   LIN {X -6.651, Y 41.522, Z 66.300}
   LaserStart_Ext()
   LIN {X -0.584, Y 41.522, Z 66.300}
   LaserEnd_Ext()
   LIN {X -0.132, Y 40.522, Z 66.300}
   LaserStart_Ext()
   LIN {X -6.592, Y 40.522, Z 66.300}
   LaserEnd_Ext()
   LIN {X -6.269, Y 39.522, Z 66.300}
   LaserStart_Ext()
   LIN {X 0.315, Y 39.522, Z 66.300}
   LaserEnd_Ext()
   LIN {X 0.738, Y 38.522, Z 66.300}
   LaserStart_Ext()
   LIN {X -5.884, Y 38.522, Z 66.300}
   LaserEnd_Ext()
   LIN {X -5.510, Y 37.522, Z 66.300}
   LaserStart_Ext()
   LIN {X 1.160, Y 37.522, Z 66.300}
   LaserEnd_Ext()
   LIN {X 1.563, Y 36.522, Z 66.300}
   LaserStart_Ext()
   LIN {X -5.164, Y 36.522, Z 66.300}
   LaserEnd_Ext()
   LIN {X -4.819, Y 35.522, Z 66.300}
   LaserStart_Ext()
   LIN {X 1.943, Y 35.522, Z 66.300}
   LaserEnd_Ext()
   LIN {X 2.327, Y 34.522, Z 66.300}
   LaserStart_Ext()
   LIN {X -4.502, Y 34.522, Z 66.300}
   LaserEnd_Ext()
   LIN {X -4.196, Y 33.522, Z 66.300}
   LaserStart_Ext()
   LIN {X 2.711, Y 33.522, Z 66.300}
   LaserEnd_Ext()
   LIN {X 3.089, Y 32.522, Z 66.300}
   LaserStart_Ext()
   LIN {X -3.888, Y 32.522, Z 66.300}
   LaserEnd_Ext()
   LIN {X -3.629, Y 31.522, Z 66.300}
   LaserStart_Ext()
   LIN {X 3.434, Y 31.522, Z 66.300}
   LaserEnd_Ext()
   LIN {X 3.759, Y 30.522, Z 66.300}
   LaserStart_Ext()
   LIN {X -3.371, Y 30.522, Z 66.300}
   LaserEnd_Ext()
   LIN {X -3.113, Y 29.522, Z 66.300}
   LaserStart_Ext()
   LIN {X 4.082, Y 29.522, Z 66.300}
   LaserEnd_Ext()
   LIN {X 4.405, Y 28.522, Z 66.300}
   LaserStart_Ext()
   LIN {X -2.876, Y 28.522, Z 66.300}
   LaserEnd_Ext()
   LIN {X -2.680, Y 27.522, Z 66.300}
   LaserStart_Ext()
   LIN {X 4.728, Y 27.522, Z 66.300}
   LaserEnd_Ext()
   LIN {X 5.051, Y 26.522, Z 66.300}
   LaserStart_Ext()
   LIN {X -2.482, Y 26.522, Z 66.300}
   LaserEnd_Ext()
   LIN {X -2.285, Y 25.522, Z 66.300}
   LaserStart_Ext()
   LIN {X 5.305, Y 25.522, Z 66.300}
   LaserEnd_Ext()
   LIN {X 5.559, Y 24.522, Z 66.300}
   LaserStart_Ext()
   LIN {X -2.087, Y 24.522, Z 66.300}
   LaserEnd_Ext()
   LIN {X -1.950, Y 23.522, Z 66.300}
   LaserStart_Ext()
   LIN {X 5.812, Y 23.522, Z 66.300}
   LaserEnd_Ext()
   LIN {X 6.066, Y 22.522, Z 66.300}
   LaserStart_Ext()
   LIN {X -1.864, Y 22.522, Z 66.300}
   LaserEnd_Ext()
   LIN {X -1.779, Y 21.522, Z 66.300}
   LaserStart_Ext()
   LIN {X 6.319, Y 21.522, Z 66.300}
   LaserEnd_Ext()
   LIN {X 6.573, Y 20.522, Z 66.300}
   LaserStart_Ext()
   LIN {X -1.694, Y 20.522, Z 66.300}
   LaserEnd_Ext()
   LIN {X -1.588, Y 19.522, Z 66.300}
   LaserStart_Ext()
   LIN {X 6.833, Y 19.522, Z 66.300}
   LaserEnd_Ext()
   LIN {X 7.071, Y 18.522, Z 66.300}
   LaserStart_Ext()
   LIN {X -1.481, Y 18.522, Z 66.300}
   LaserEnd_Ext()
   LIN {X -1.375, Y 17.522, Z 66.300}
   LaserStart_Ext()
   LIN {X 7.250, Y 17.522, Z 66.300}
   LaserEnd_Ext()
   LIN {X 7.405, Y 16.522, Z 66.300}
   LaserStart_Ext()
   LIN {X -1.269, Y 16.522, Z 66.300}
   LaserEnd_Ext()
   LIN {X -1.163, Y 15.522, Z 66.300}
   LaserStart_Ext()
   LIN {X 7.561, Y 15.522, Z 66.300}
   LaserEnd_Ext()
   LIN {X 7.716, Y 14.522, Z 66.300}
   LaserStart_Ext()
   LIN {X -1.142, Y 14.522, Z 66.300}
   LaserEnd_Ext()
   LIN {X -1.150, Y 13.522, Z 66.300}
   LaserStart_Ext()
   LIN {X 7.872, Y 13.522, Z 66.300}
   LaserEnd_Ext()
   LIN {X 8.027, Y 12.522, Z 66.300}
   LaserStart_Ext()
   LIN {X -1.158, Y 12.522, Z 66.300}
   LaserEnd_Ext()
   LIN {X -1.166, Y 11.522, Z 66.300}
   LaserStart_Ext()
   LIN {X 8.183, Y 11.522, Z 66.300}
   LaserEnd_Ext()
   LIN {X 8.339, Y 10.522, Z 66.300}
   LaserStart_Ext()
   LIN {X -1.175, Y 10.522, Z 66.300}
   LaserEnd_Ext()
   LIN {X -1.191, Y 9.522, Z 66.300}
   LaserStart_Ext()
   LIN {X 8.494, Y 9.522, Z 66.300}
   LaserEnd_Ext()
   LIN {X 8.650, Y 8.522, Z 66.300}
   LaserStart_Ext()
   LIN {X -1.230, Y 8.522, Z 66.300}
   LaserEnd_Ext()
   LIN {X -1.268, Y 7.522, Z 66.300}
   LaserStart_Ext()
   LIN {X 8.806, Y 7.522, Z 66.300}
   LaserEnd_Ext()
   LIN {X 8.956, Y 6.522, Z 66.300}
   LaserStart_Ext()
   LIN {X -1.307, Y 6.522, Z 66.300}
   LaserEnd_Ext()
   LIN {X -1.345, Y 5.522, Z 66.300}
   LaserStart_Ext()
   LIN {X 9.069, Y 5.522, Z 66.300}
   LaserEnd_Ext()
   LIN {X 9.141, Y 4.522, Z 66.300}
   LaserStart_Ext()
   LIN {X -1.463, Y 4.522, Z 66.300}
   LaserEnd_Ext()
   LIN {X -1.598, Y 3.522, Z 66.300}
   LaserStart_Ext()
   LIN {X 9.202, Y 3.522, Z 66.300}
   LaserEnd_Ext()
   LIN {X 9.264, Y 2.522, Z 66.300}
   LaserStart_Ext()
   LIN {X -1.733, Y 2.522, Z 66.300}
   LaserEnd_Ext()
   LIN {X -1.868, Y 1.522, Z 66.300}
   LaserStart_Ext()
   LIN {X 9.325, Y 1.522, Z 66.300}
   LaserEnd_Ext()
   LIN {X 9.387, Y 0.522, Z 66.300}
   LaserStart_Ext()
   LIN {X -2.004, Y 0.522, Z 66.300}
   LaserEnd_Ext()
   LIN {X -2.141, Y -0.478, Z 66.300}
   LaserStart_Ext()
   LIN {X 9.437, Y -0.478, Z 66.300}
   LaserEnd_Ext()
   LIN {X 9.443, Y -1.478, Z 66.300}
   LaserStart_Ext()
   LIN {X -2.360, Y -1.478, Z 66.300}
   LaserEnd_Ext()
   LIN {X -2.584, Y -2.478, Z 66.300}
   LaserStart_Ext()
   LIN {X 9.450, Y -2.478, Z 66.300}
   LaserEnd_Ext()
   LIN {X 9.459, Y -3.478, Z 66.300}
   LaserStart_Ext()
   LIN {X -2.803, Y -3.478, Z 66.300}
   LaserEnd_Ext()
   LIN {X -3.022, Y -4.478, Z 66.300}
   LaserStart_Ext()
   LIN {X 9.468, Y -4.478, Z 66.300}
   LaserEnd_Ext()
   LIN {X 9.477, Y -5.478, Z 66.300}
   LaserStart_Ext()
   LIN {X -3.241, Y -5.478, Z 66.300}
   LaserEnd_Ext()
   LIN {X -3.460, Y -6.478, Z 66.300}
   LaserStart_Ext()
   LIN {X 9.486, Y -6.478, Z 66.300}
   LaserEnd_Ext()
   LIN {X 9.460, Y -7.478, Z 66.300}
   LaserStart_Ext()
   LIN {X -3.732, Y -7.478, Z 66.300}
   LaserEnd_Ext()
   LIN {X -4.029, Y -8.478, Z 66.300}
   LaserStart_Ext()
   LIN {X 9.419, Y -8.478, Z 66.300}
   LaserEnd_Ext()
   LIN {X 9.374, Y -9.478, Z 66.300}
   LaserStart_Ext()
   LIN {X -4.322, Y -9.478, Z 66.300}
   LaserEnd_Ext()
   LIN {X -4.616, Y -10.478, Z 66.300}
   LaserStart_Ext()
   LIN {X 9.329, Y -10.478, Z 66.300}
   LaserEnd_Ext()
   LIN {X 9.284, Y -11.478, Z 66.300}
   LaserStart_Ext()
   LIN {X -4.963, Y -11.478, Z 66.300}
   LaserEnd_Ext()
   LIN {X -5.315, Y -12.478, Z 66.300}
   LaserStart_Ext()
   LIN {X 9.205, Y -12.478, Z 66.300}
   LaserEnd_Ext()
   LIN {X 9.125, Y -13.478, Z 66.300}
   LaserStart_Ext()
   LIN {X -5.670, Y -13.478, Z 66.300}
   LaserEnd_Ext()
   LIN {X -6.040, Y -14.478, Z 66.300}
   LaserStart_Ext()
   LIN {X -1.258, Y -14.478, Z 66.300}
   LaserEnd_Ext()
   LIN {X 2.231, Y -14.478, Z 66.300}
   LaserStart_Ext()
   LIN {X 9.041, Y -14.478, Z 66.300}
   LaserEnd_Ext()
   LIN {X 8.948, Y -15.478, Z 66.300}
   LaserStart_Ext()
   LIN {X 3.969, Y -15.478, Z 66.300}
   LaserEnd_Ext()
   LIN {X -3.325, Y -15.478, Z 66.300}
   LaserStart_Ext()
   LIN {X -6.451, Y -15.478, Z 66.300}
   LaserEnd_Ext()
   LIN {X -6.857, Y -16.478, Z 66.300}
   LaserStart_Ext()
   LIN {X -4.408, Y -16.478, Z 66.300}
   LaserEnd_Ext()
   LIN {X 4.864, Y -16.478, Z 66.300}
   LaserStart_Ext()
   LIN {X 8.833, Y -16.478, Z 66.300}
   LaserEnd_Ext()
   LIN {X 8.720, Y -17.478, Z 66.300}
   LaserStart_Ext()
   LIN {X 5.511, Y -17.478, Z 66.300}
   LaserEnd_Ext()
   LIN {X -4.909, Y -17.478, Z 66.300}
   LaserStart_Ext()
   LIN {X -7.170, Y -17.478, Z 66.300}
   LaserEnd_Ext()
   LIN {X -7.405, Y -18.478, Z 66.300}
   LaserStart_Ext()
   LIN {X -5.231, Y -18.478, Z 66.300}
   LaserEnd_Ext()
   LIN {X 6.029, Y -18.478, Z 66.300}
   LaserStart_Ext()
   LIN {X 8.601, Y -18.478, Z 66.300}
   LaserEnd_Ext()
   LIN {X 8.461, Y -19.478, Z 66.300}
   LaserStart_Ext()
   LIN {X 6.119, Y -19.478, Z 66.300}
   LaserEnd_Ext()
   LIN {X -5.554, Y -19.478, Z 66.300}
   LaserStart_Ext()
   LIN {X -7.643, Y -19.478, Z 66.300}
   LaserEnd_Ext()
   LIN {X -7.604, Y -20.478, Z 66.300}
   LaserStart_Ext()
   LIN {X -5.694, Y -20.478, Z 66.300}
   LaserEnd_Ext()
   LIN {X 6.211, Y -20.478, Z 66.300}
   LaserStart_Ext()
   LIN {X 8.319, Y -20.478, Z 66.300}
   LaserEnd_Ext()
   LIN {X 8.137, Y -21.478, Z 66.300}
   LaserStart_Ext()
   LIN {X 6.041, Y -21.478, Z 66.300}
   LaserEnd_Ext()
   LIN {X -5.485, Y -21.478, Z 66.300}
   LaserStart_Ext()
   LIN {X -7.453, Y -21.478, Z 66.300}
   LaserEnd_Ext()
   LIN {X -7.299, Y -22.478, Z 66.300}
   LaserStart_Ext()
   LIN {X -5.273, Y -22.478, Z 66.300}
   LaserEnd_Ext()
   LIN {X 5.653, Y -22.478, Z 66.300}
   LaserStart_Ext()
   LIN {X 7.806, Y -22.478, Z 66.300}
   LaserEnd_Ext()
   LIN {X 7.474, Y -23.478, Z 66.300}
   LaserStart_Ext()
   LIN {X 5.253, Y -23.478, Z 66.300}
   LaserEnd_Ext()
   LIN {X -4.630, Y -23.478, Z 66.300}
   LaserStart_Ext()
   LIN {X -6.924, Y -23.478, Z 66.300}
   LaserEnd_Ext()
   LIN {X -6.279, Y -24.478, Z 66.300}
   LaserStart_Ext()
   LIN {X -3.896, Y -24.478, Z 66.300}
   LaserEnd_Ext()
   LIN {X 4.265, Y -24.478, Z 66.300}
   LaserStart_Ext()
   LIN {X 6.808, Y -24.478, Z 66.300}
   LaserEnd_Ext()
   LIN {X 5.993, Y -25.478, Z 66.300}
   LaserStart_Ext()
   LIN {X 2.928, Y -25.478, Z 66.300}
   LaserEnd_Ext()
   LIN {X -2.348, Y -25.478, Z 66.300}
   LaserStart_Ext()
   LIN {X -5.639, Y -25.478, Z 66.300}
   LaserEnd_Ext()
   LIN {X -4.529, Y -26.478, Z 66.300}
   LaserStart_Ext()
   LIN {X 5.068, Y -26.478, Z 66.300}
   LaserEnd_Ext()
   LIN {X 3.258, Y -27.478, Z 66.300}
   LaserStart_Ext()
   LIN {X -2.674, Y -27.478, Z 66.300}
   LaserEnd_Ext()
   LIN {X 5.111, Y -18.522, Z 67.150}
   LaserStart_Ext()
   LIN {X 5.164, Y -19.081, Z 67.150} C_DIS
   LIN {X 5.316, Y -20.722, Z 67.150} C_DIS
   LIN {X 4.744, Y -22.209, Z 67.150} C_DIS
   LIN {X 4.460, Y -22.939, Z 67.150} C_DIS
   LIN {X 3.234, Y -24.097, Z 67.150} C_DIS
   LIN {X 2.927, Y -24.388, Z 67.150} C_DIS
   LIN {X 2.658, Y -24.480, Z 67.150} C_DIS
   LIN {X 0.847, Y -25.087, Z 67.150} C_DIS
   LIN {X -0.754, Y -24.932, Z 67.150} C_DIS
   LIN {X -1.190, Y -24.888, Z 67.150} C_DIS
   LIN {X -1.701, Y -24.596, Z 67.150} C_DIS
   LIN {X -2.985, Y -23.865, Z 67.150} C_DIS
   LIN {X -3.728, Y -22.861, Z 67.150} C_DIS
   LIN {X -4.221, Y -22.189, Z 67.150} C_DIS
   LIN {X -4.389, Y -21.390, Z 67.150} C_DIS
   LIN {X -4.654, Y -20.148, Z 67.150} C_DIS
   LIN {X -4.025, Y -18.200, Z 67.150} C_DIS
   LIN {X -3.718, Y -17.225, Z 67.150} C_DIS
   LIN {X -2.185, Y -15.809, Z 67.150} C_DIS
   LIN {X -0.151, Y -15.135, Z 67.150} C_DIS
   LIN {X 1.590, Y -15.303, Z 67.150} C_DIS
   LIN {X 1.882, Y -15.330, Z 67.150} C_DIS
   LIN {X 2.218, Y -15.522, Z 67.150} C_DIS
   LIN {X 3.724, Y -16.390, Z 67.150} C_DIS
   LIN {X 4.736, Y -17.949, Z 67.150} C_DIS
   LIN {X 5.111, Y -18.522, Z 67.150}
   LaserEnd_Ext()
   LIN {X -3.141, Y -0.519, Z 67.150}
   LaserStart_Ext()
   LIN {X -4.458, Y -6.534, Z 67.150} C_DIS
   LIN {X -4.638, Y -7.154, Z 67.150} C_DIS
   LIN {X -5.541, Y -10.227, Z 67.150} C_DIS
   LIN {X -6.686, Y -13.482, Z 67.150} C_DIS
   LIN {X -6.815, Y -13.852, Z 67.150} C_DIS
   LIN {X -6.899, Y -14.062, Z 67.150} C_DIS
   LIN {X -7.931, Y -16.604, Z 67.150} C_DIS
   LIN {X -8.614, Y -19.534, Z 67.150} C_DIS
   LIN {X -8.652, Y -19.692, Z 67.150} C_DIS
   LIN {X -8.620, Y -19.900, Z 67.150} C_DIS
   LIN {X -8.083, Y -23.358, Z 67.150} C_DIS
   LIN {X -6.321, Y -26.092, Z 67.150} C_DIS
   LIN {X -6.049, Y -26.508, Z 67.150} C_DIS
   LIN {X -5.702, Y -26.754, Z 67.150} C_DIS
   LIN {X -3.685, Y -28.200, Z 67.150} C_DIS
   LIN {X -1.505, Y -28.715, Z 67.150} C_DIS
   LIN {X 0.077, Y -29.119, Z 67.150} C_DIS
   LIN {X 2.778, Y -28.726, Z 67.150} C_DIS
   LIN {X 3.131, Y -28.668, Z 67.150} C_DIS
   LIN {X 3.388, Y -28.528, Z 67.150} C_DIS
   LIN {X 6.099, Y -27.012, Z 67.150} C_DIS
   LIN {X 7.842, Y -24.873, Z 67.150} C_DIS
   LIN {X 8.337, Y -24.241, Z 67.150} C_DIS
   LIN {X 8.664, Y -23.241, Z 67.150} C_DIS
   LIN {X 9.265, Y -21.428, Z 67.150} C_DIS
   LIN {X 9.444, Y -20.170, Z 67.150} C_DIS
   LIN {X 9.713, Y -18.195, Z 67.150} C_DIS
   LIN {X 10.022, Y -15.403, Z 67.150} C_DIS
   LIN {X 10.039, Y -15.252, Z 67.150} C_DIS
   LIN {X 10.049, Y -15.138, Z 67.150} C_DIS
   LIN {X 10.342, Y -11.458, Z 67.150} C_DIS
   LIN {X 10.422, Y -9.675, Z 67.150} C_DIS
   LIN {X 10.536, Y -6.674, Z 67.150} C_DIS
   LIN {X 10.491, Y -1.605, Z 67.150} C_DIS
   LIN {X 10.468, Y -0.160, Z 67.150} C_DIS
   LIN {X 10.251, Y 3.362, Z 67.150} C_DIS
   LIN {X 10.173, Y 4.620, Z 67.150} C_DIS
   LIN {X 10.143, Y 5.122, Z 67.150} C_DIS
   LIN {X 9.922, Y 7.075, Z 67.150} C_DIS
   LIN {X 8.378, Y 16.995, Z 67.150} C_DIS
   LIN {X 7.939, Y 19.269, Z 67.150} C_DIS
   LIN {X 7.156, Y 22.245, Z 67.150} C_DIS
   LIN {X 6.006, Y 26.781, Z 67.150} C_DIS
   LIN {X 4.979, Y 29.959, Z 67.150} C_DIS
   LIN {X 4.276, Y 32.119, Z 67.150} C_DIS
   LIN {X 3.714, Y 33.661, Z 67.150} C_DIS
   LIN {X 2.866, Y 35.872, Z 67.150} C_DIS
   LIN {X 2.282, Y 37.356, Z 67.150} C_DIS
   LIN {X 1.333, Y 39.592, Z 67.150} C_DIS
   LIN {X 1.196, Y 39.917, Z 67.150} C_DIS
   LIN {X 1.126, Y 40.074, Z 67.150} C_DIS
   LIN {X 0.410, Y 41.666, Z 67.150} C_DIS
   LIN {X -0.110, Y 42.781, Z 67.150} C_DIS
   LIN {X -0.218, Y 43.011, Z 67.150} C_DIS
   LIN {X -0.443, Y 43.320, Z 67.150} C_DIS
   LIN {X -1.082, Y 44.201, Z 67.150} C_DIS
   LIN {X -1.717, Y 44.585, Z 67.150} C_DIS
   LIN {X -2.573, Y 45.098, Z 67.150} C_DIS
   LIN {X -4.184, Y 45.264, Z 67.150} C_DIS
   LIN {X -4.309, Y 45.277, Z 67.150} C_DIS
   LIN {X -6.474, Y 44.269, Z 67.150} C_DIS
   LIN {X -6.615, Y 44.145, Z 67.150} C_DIS
   LIN {X -7.543, Y 42.764, Z 67.150} C_DIS
   LIN {X -7.760, Y 41.294, Z 67.150} C_DIS
   LIN {X -7.798, Y 41.016, Z 67.150} C_DIS
   LIN {X -7.735, Y 40.758, Z 67.150} C_DIS
   LIN {X -7.502, Y 39.809, Z 67.150} C_DIS
   LIN {X -7.222, Y 39.097, Z 67.150} C_DIS
   LIN {X -7.045, Y 38.645, Z 67.150} C_DIS
   LIN {X -6.784, Y 37.952, Z 67.150} C_DIS
   LIN {X -6.479, Y 37.149, Z 67.150} C_DIS
   LIN {X -6.105, Y 36.074, Z 67.150} C_DIS
   LIN {X -5.702, Y 34.909, Z 67.150} C_DIS
   LIN {X -5.602, Y 34.578, Z 67.150} C_DIS
   LIN {X -4.875, Y 32.225, Z 67.150} C_DIS
   LIN {X -4.185, Y 29.550, Z 67.150} C_DIS
   LIN {X -3.922, Y 28.545, Z 67.150} C_DIS
   LIN {X -3.696, Y 27.417, Z 67.150} C_DIS
   LIN {X -3.001, Y 23.898, Z 67.150} C_DIS
   LIN {X -2.805, Y 21.594, Z 67.150} C_DIS
   LIN {X -2.151, Y 15.433, Z 67.150} C_DIS
   LIN {X -2.203, Y 9.073, Z 67.150} C_DIS
   LIN {X -2.350, Y 5.267, Z 67.150} C_DIS
   LIN {X -3.104, Y -0.321, Z 67.150} C_DIS
   LIN {X -3.141, Y -0.519, Z 67.150}
   LaserEnd_Ext()
   LIN {X -7.280, Y -22.014, Z 67.150}
   LaserStart_Ext()
   LIN {X -7.280, Y -18.216, Z 67.150}
   LaserEnd_Ext()
   LIN {X -6.280, Y 42.851, Z 67.150}
   LaserStart_Ext()
   LIN {X -6.280, Y 39.434, Z 67.150}
   LaserEnd_Ext()
   LIN {X -6.280, Y -15.196, Z 67.150}
   LaserStart_Ext()
   LIN {X -6.280, Y -24.309, Z 67.150}
   LaserEnd_Ext()
   LIN {X -5.280, Y -25.827, Z 67.150}
   LaserStart_Ext()
   LIN {X -5.280, Y -22.014, Z 67.150}
   LaserEnd_Ext()
   LIN {X -5.280, Y -18.831, Z 67.150}
   LaserStart_Ext()
   LIN {X -5.280, Y -12.498, Z 67.150}
   LaserEnd_Ext()
   LIN {X -5.280, Y 36.745, Z 67.150}
   LaserStart_Ext()
   LIN {X -5.280, Y 43.722, Z 67.150}
   LaserEnd_Ext()
   LIN {X -4.280, Y 44.189, Z 67.150}
   LaserStart_Ext()
   LIN {X -4.280, Y 33.686, Z 67.150}
   LaserEnd_Ext()
   LIN {X -4.280, Y -9.483, Z 67.150}
   LaserStart_Ext()
   LIN {X -4.280, Y -16.383, Z 67.150}
   LaserEnd_Ext()
   LIN {X -4.280, Y -23.796, Z 67.150}
   LaserStart_Ext()
   LIN {X -4.280, Y -26.543, Z 67.150}
   LaserEnd_Ext()
   LIN {X -3.280, Y -27.260, Z 67.150}
   LaserStart_Ext()
   LIN {X -3.280, Y -24.848, Z 67.150}
   LaserEnd_Ext()
   LIN {X -3.280, Y -15.459, Z 67.150}
   LaserStart_Ext()
   LIN {X -3.280, Y -5.827, Z 67.150}
   LaserEnd_Ext()
   LIN {X -3.280, Y 30.045, Z 67.150}
   LaserStart_Ext()
   LIN {X -3.280, Y 44.165, Z 67.150}
   LaserEnd_Ext()
   LIN {X -2.280, Y 43.756, Z 67.150}
   LaserStart_Ext()
   LIN {X -2.280, Y 25.405, Z 67.150}
   LaserEnd_Ext()
   LIN {X -2.280, Y -1.261, Z 67.150}
   LaserStart_Ext()
   LIN {X -2.280, Y -14.787, Z 67.150}
   LaserEnd_Ext()
   LIN {X -2.280, Y -25.417, Z 67.150}
   LaserStart_Ext()
   LIN {X -2.280, Y -27.505, Z 67.150}
   LaserEnd_Ext()
   LIN {X -1.280, Y -27.741, Z 67.150}
   LaserStart_Ext()
   LIN {X -1.280, Y -25.884, Z 67.150}
   LaserEnd_Ext()
   LIN {X -1.280, Y -14.456, Z 67.150}
   LaserStart_Ext()
   LIN {X -1.280, Y 7.058, Z 67.150}
   LaserEnd_Ext()
   LIN {X -1.280, Y 16.700, Z 67.150}
   LaserStart_Ext()
   LIN {X -1.280, Y 42.771, Z 67.150}
   LaserEnd_Ext()
   LIN {X -0.280, Y 40.762, Z 67.150}
   LaserStart_Ext()
   LIN {X -0.280, Y -14.144, Z 67.150}
   LaserEnd_Ext()
   LIN {X -0.280, Y -25.983, Z 67.150}
   LaserStart_Ext()
   LIN {X -0.280, Y -27.996, Z 67.150}
   LaserEnd_Ext()
   LIN {X 0.720, Y -28.015, Z 67.150}
   LaserStart_Ext()
   LIN {X 0.720, Y -26.079, Z 67.150}
   LaserEnd_Ext()
   LIN {X 0.720, Y -14.215, Z 67.150}
   LaserStart_Ext()
   LIN {X 0.720, Y 38.477, Z 67.150}
   LaserEnd_Ext()
   LIN {X 1.720, Y 36.053, Z 67.150}
   LaserStart_Ext()
   LIN {X 1.720, Y -14.311, Z 67.150}
   LaserEnd_Ext()
   LIN {X 1.720, Y -25.849, Z 67.150}
   LaserStart_Ext()
   LIN {X 1.720, Y -27.869, Z 67.150}
   LaserEnd_Ext()
   LIN {X 2.720, Y -27.722, Z 67.150}
   LaserStart_Ext()
   LIN {X 2.720, Y -25.514, Z 67.150}
   LaserEnd_Ext()
   LIN {X 2.720, Y -14.658, Z 67.150}
   LaserStart_Ext()
   LIN {X 2.720, Y 33.461, Z 67.150}
   LaserEnd_Ext()
   LIN {X 3.720, Y 30.595, Z 67.150}
   LaserStart_Ext()
   LIN {X 3.720, Y -15.234, Z 67.150}
   LaserEnd_Ext()
   LIN {X 3.720, Y -25.014, Z 67.150}
   LaserStart_Ext()
   LIN {X 3.720, Y -27.197, Z 67.150}
   LaserEnd_Ext()
   LIN {X 4.720, Y -26.638, Z 67.150}
   LaserStart_Ext()
   LIN {X 4.720, Y -24.069, Z 67.150}
   LaserEnd_Ext()
   LIN {X 4.720, Y -16.088, Z 67.150}
   LaserStart_Ext()
   LIN {X 4.720, Y 27.507, Z 67.150}
   LaserEnd_Ext()
   LIN {X 5.720, Y 23.839, Z 67.150}
   LaserStart_Ext()
   LIN {X 5.720, Y -17.626, Z 67.150}
   LaserEnd_Ext()
   LIN {X 5.720, Y -22.457, Z 67.150}
   LaserStart_Ext()
   LIN {X 5.720, Y -25.894, Z 67.150}
   LaserEnd_Ext()
   LIN {X 6.720, Y -24.667, Z 67.150}
   LaserStart_Ext()
   LIN {X 6.720, Y 19.972, Z 67.150}
   LaserEnd_Ext()
   LIN {X 7.720, Y 14.721, Z 67.150}
   LaserStart_Ext()
   LIN {X 7.720, Y -22.909, Z 67.150}
   LaserEnd_Ext()
   LIN {X 8.720, Y -18.075, Z 67.150}
   LaserStart_Ext()
   LIN {X 8.720, Y 8.294, Z 67.150}
   LaserEnd_Ext()
   LIN {X -4.138, Y -22.147, Z 68.000}
   LaserStart_Ext()
   LIN {X -4.289, Y -21.447, Z 68.000} C_DIS
   LIN {X -4.575, Y -20.106, Z 68.000} C_DIS
   LIN {X -4.291, Y -19.226, Z 68.000} C_DIS
   LIN {X -3.647, Y -17.183, Z 68.000} C_DIS
   LIN {X -2.794, Y -16.395, Z 68.000} C_DIS
   LIN {X -2.090, Y -15.746, Z 68.000} C_DIS
   LIN {X -0.721, Y -15.295, Z 68.000} C_DIS
   LIN {X -0.083, Y -15.083, Z 68.000} C_DIS
   LIN {X 0.376, Y -15.128, Z 68.000} C_DIS
   LIN {X 1.950, Y -15.273, Z 68.000} C_DIS
   LIN {X 3.753, Y -16.305, Z 68.000} C_DIS
   LIN {X 5.186, Y -18.457, Z 68.000} C_DIS
   LIN {X 5.381, Y -20.496, Z 68.000} C_DIS
   LIN {X 5.396, Y -20.658, Z 68.000} C_DIS
   LIN {X 5.029, Y -21.613, Z 68.000} C_DIS
   LIN {X 4.542, Y -22.882, Z 68.000} C_DIS
   LIN {X 4.408, Y -23.009, Z 68.000} C_DIS
   LIN {X 3.019, Y -24.327, Z 68.000} C_DIS
   LIN {X 1.507, Y -24.842, Z 68.000} C_DIS
   LIN {X 0.938, Y -25.032, Z 68.000} C_DIS
   LIN {X 0.103, Y -24.952, Z 68.000} C_DIS
   LIN {X -1.100, Y -24.839, Z 68.000} C_DIS
   LIN {X -1.883, Y -24.396, Z 68.000} C_DIS
   LIN {X -2.897, Y -23.820, Z 68.000} C_DIS
   LIN {X -3.721, Y -22.706, Z 68.000} C_DIS
   LIN {X -4.138, Y -22.147, Z 68.000}
   LaserEnd_Ext()
   LIN {X -6.748, Y 37.749, Z 68.000}
   LaserStart_Ext()
   LIN {X -6.535, Y 37.185, Z 68.000} C_DIS
   LIN {X -6.212, Y 36.259, Z 68.000} C_DIS
   LIN {X -5.752, Y 34.948, Z 68.000} C_DIS
   LIN {X -5.394, Y 33.799, Z 68.000} C_DIS
   LIN {X -4.903, Y 32.210, Z 68.000} C_DIS
   LIN {X -4.601, Y 31.041, Z 68.000} C_DIS
   LIN {X -3.931, Y 28.480, Z 68.000} C_DIS
   LIN {X -3.357, Y 25.605, Z 68.000} C_DIS
   LIN {X -3.016, Y 23.882, Z 68.000} C_DIS
   LIN {X -2.920, Y 22.754, Z 68.000} C_DIS
   LIN {X -2.166, Y 15.650, Z 68.000} C_DIS
   LIN {X -2.226, Y 8.314, Z 68.000} C_DIS
   LIN {X -2.349, Y 5.105, Z 68.000} C_DIS
   LIN {X -2.986, Y 0.394, Z 68.000} C_DIS
   LIN {X -3.161, Y -0.794, Z 68.000} C_DIS
   LIN {X -3.456, Y -2.131, Z 68.000} C_DIS
   LIN {X -4.411, Y -6.490, Z 68.000} C_DIS
   LIN {X -5.183, Y -9.160, Z 68.000} C_DIS
   LIN {X -5.485, Y -10.187, Z 68.000} C_DIS
   LIN {X -5.867, Y -11.274, Z 68.000} C_DIS
   LIN {X -6.748, Y -13.809, Z 68.000} C_DIS
   LIN {X -7.326, Y -15.254, Z 68.000} C_DIS
   LIN {X -7.860, Y -16.570, Z 68.000} C_DIS
   LIN {X -8.253, Y -18.255, Z 68.000} C_DIS
   LIN {X -8.574, Y -19.660, Z 68.000} C_DIS
   LIN {X -8.331, Y -21.172, Z 68.000} C_DIS
   LIN {X -7.996, Y -23.325, Z 68.000} C_DIS
   LIN {X -7.009, Y -24.856, Z 68.000} C_DIS
   LIN {X -5.955, Y -26.469, Z 68.000} C_DIS
   LIN {X -4.613, Y -27.421, Z 68.000} C_DIS
   LIN {X -3.588, Y -28.156, Z 68.000} C_DIS
   LIN {X -2.480, Y -28.418, Z 68.000} C_DIS
   LIN {X 0.041, Y -29.062, Z 68.000} C_DIS
   LIN {X 2.330, Y -28.729, Z 68.000} C_DIS
   LIN {X 3.173, Y -28.627, Z 68.000} C_DIS
   LIN {X 4.698, Y -27.761, Z 68.000} C_DIS
   LIN {X 6.274, Y -26.880, Z 68.000} C_DIS
   LIN {X 7.075, Y -25.896, Z 68.000} C_DIS
   LIN {X 8.426, Y -24.168, Z 68.000} C_DIS
   LIN {X 9.319, Y -21.437, Z 68.000} C_DIS
   LIN {X 9.355, Y -21.295, Z 68.000} C_DIS
   LIN {X 9.788, Y -18.120, Z 68.000} C_DIS
   LIN {X 9.988, Y -16.311, Z 68.000} C_DIS
   LIN {X 10.107, Y -15.176, Z 68.000} C_DIS
   LIN {X 10.374, Y -11.711, Z 68.000} C_DIS
   LIN {X 10.400, Y -11.382, Z 68.000} C_DIS
   LIN {X 10.407, Y -11.239, Z 68.000} C_DIS
   LIN {X 10.584, Y -6.597, Z 68.000} C_DIS
   LIN {X 10.558, Y -3.758, Z 68.000} C_DIS
   LIN {X 10.500, Y -0.083, Z 68.000} C_DIS
   LIN {X 10.337, Y 2.556, Z 68.000} C_DIS
   LIN {X 10.237, Y 4.187, Z 68.000} C_DIS
   LIN {X 10.197, Y 4.837, Z 68.000} C_DIS
   LIN {X 9.911, Y 7.370, Z 68.000} C_DIS
   LIN {X 8.582, Y 15.907, Z 68.000} C_DIS
   LIN {X 7.902, Y 19.435, Z 68.000} C_DIS
   LIN {X 6.686, Y 24.053, Z 68.000} C_DIS
   LIN {X 5.996, Y 26.772, Z 68.000} C_DIS
   LIN {X 5.381, Y 28.678, Z 68.000} C_DIS
   LIN {X 4.335, Y 31.887, Z 68.000} C_DIS
   LIN {X 3.636, Y 33.809, Z 68.000} C_DIS
   LIN {X 3.522, Y 34.123, Z 68.000} C_DIS
   LIN {X 3.195, Y 34.950, Z 68.000} C_DIS
   LIN {X 2.226, Y 37.413, Z 68.000} C_DIS
   LIN {X 1.906, Y 38.169, Z 68.000} C_DIS
   LIN {X 1.134, Y 39.972, Z 68.000} C_DIS
   LIN {X 0.430, Y 41.531, Z 68.000} C_DIS
   LIN {X 0.344, Y 41.719, Z 68.000} C_DIS
   LIN {X 0.234, Y 41.954, Z 68.000} C_DIS
   LIN {X -0.287, Y 43.062, Z 68.000} C_DIS
   LIN {X -0.767, Y 43.723, Z 68.000} C_DIS
   LIN {X -1.154, Y 44.251, Z 68.000} C_DIS
   LIN {X -2.049, Y 44.785, Z 68.000} C_DIS
   LIN {X -2.647, Y 45.144, Z 68.000} C_DIS
   LIN {X -3.093, Y 45.190, Z 68.000} C_DIS
   LIN {X -4.383, Y 45.319, Z 68.000} C_DIS
   LIN {X -5.484, Y 44.806, Z 68.000} C_DIS
   LIN {X -6.689, Y 44.204, Z 68.000} C_DIS
   LIN {X -7.456, Y 43.070, Z 68.000} C_DIS
   LIN {X -7.574, Y 42.894, Z 68.000} C_DIS
   LIN {X -7.613, Y 42.634, Z 68.000} C_DIS
   LIN {X -7.867, Y 41.136, Z 68.000} C_DIS
   LIN {X -7.594, Y 39.967, Z 68.000} C_DIS
   LIN {X -7.564, Y 39.844, Z 68.000} C_DIS
   LIN {X -7.504, Y 39.692, Z 68.000} C_DIS
   LIN {X -7.104, Y 38.681, Z 68.000} C_DIS
   LIN {X -6.748, Y 37.749, Z 68.000}
   LaserEnd_Ext()
   LIN {X -2.609, Y -27.360, Z 68.000}
   LaserStart_Ext()
   LIN {X 3.379, Y -27.360, Z 68.000}
   LaserEnd_Ext()
   LIN {X 5.154, Y -26.360, Z 68.000}
   LaserStart_Ext()
   LIN {X -4.380, Y -26.360, Z 68.000}
   LaserEnd_Ext()
   LIN {X -5.485, Y -25.360, Z 68.000}
   LaserStart_Ext()
   LIN {X -2.210, Y -25.360, Z 68.000}
   LaserEnd_Ext()
   LIN {X 3.087, Y -25.360, Z 68.000}
   LaserStart_Ext()
   LIN {X 6.222, Y -25.360, Z 68.000}
   LaserEnd_Ext()
   LIN {X 7.006, Y -24.360, Z 68.000}
   LaserStart_Ext()
   LIN {X 4.437, Y -24.360, Z 68.000}
   LaserEnd_Ext()
   LIN {X -3.741, Y -24.360, Z 68.000}
   LaserStart_Ext()
   LIN {X -6.139, Y -24.360, Z 68.000}
   LaserEnd_Ext()
   LIN {X -6.784, Y -23.360, Z 68.000}
   LaserStart_Ext()
   LIN {X -4.481, Y -23.360, Z 68.000}
   LaserEnd_Ext()
   LIN {X 5.419, Y -23.360, Z 68.000}
   LaserStart_Ext()
   LIN {X 7.638, Y -23.360, Z 68.000}
   LaserEnd_Ext()
   LIN {X 7.965, Y -22.360, Z 68.000}
   LaserStart_Ext()
   LIN {X 5.813, Y -22.360, Z 68.000}
   LaserEnd_Ext()
   LIN {X -5.115, Y -22.360, Z 68.000}
   LaserStart_Ext()
   LIN {X -7.134, Y -22.360, Z 68.000}
   LaserEnd_Ext()
   LIN {X -7.290, Y -21.360, Z 68.000}
   LaserStart_Ext()
   LIN {X -5.330, Y -21.360, Z 68.000}
   LaserEnd_Ext()
   LIN {X 6.198, Y -21.360, Z 68.000}
   LaserStart_Ext()
   LIN {X 8.292, Y -21.360, Z 68.000}
   LaserEnd_Ext()
   LIN {X 8.473, Y -20.360, Z 68.000}
   LaserStart_Ext()
   LIN {X 6.373, Y -20.360, Z 68.000}
   LaserEnd_Ext()
   LIN {X -5.543, Y -20.360, Z 68.000}
   LaserStart_Ext()
   LIN {X -7.449, Y -20.360, Z 68.000}
   LaserEnd_Ext()
   LIN {X -7.480, Y -19.360, Z 68.000}
   LaserStart_Ext()
   LIN {X -5.385, Y -19.360, Z 68.000}
   LaserEnd_Ext()
   LIN {X 6.277, Y -19.360, Z 68.000}
   LaserStart_Ext()
   LIN {X 8.609, Y -19.360, Z 68.000}
   LaserEnd_Ext()
   LIN {X 8.746, Y -18.360, Z 68.000}
   LaserStart_Ext()
   LIN {X 6.181, Y -18.360, Z 68.000}
   LaserEnd_Ext()
   LIN {X -5.066, Y -18.360, Z 68.000}
   LaserStart_Ext()
   LIN {X -7.251, Y -18.360, Z 68.000}
   LaserEnd_Ext()
   LIN {X -7.017, Y -17.360, Z 68.000}
   LaserStart_Ext()
   LIN {X -4.751, Y -17.360, Z 68.000}
   LaserEnd_Ext()
   LIN {X 5.663, Y -17.360, Z 68.000}
   LaserStart_Ext()
   LIN {X 8.865, Y -17.360, Z 68.000}
   LaserEnd_Ext()
   LIN {X 8.976, Y -16.360, Z 68.000}
   LaserStart_Ext()
   LIN {X 5.009, Y -16.360, Z 68.000}
   LaserEnd_Ext()
   LIN {X -4.230, Y -16.360, Z 68.000}
   LaserStart_Ext()
   LIN {X -6.696, Y -16.360, Z 68.000}
   LaserEnd_Ext()
   LIN {X -6.291, Y -15.360, Z 68.000}
   LaserStart_Ext()
   LIN {X -3.146, Y -15.360, Z 68.000}
   LaserEnd_Ext()
   LIN {X 4.115, Y -15.360, Z 68.000}
   LaserStart_Ext()
   LIN {X 9.082, Y -15.360, Z 68.000}
   LaserEnd_Ext()
   LIN {X 9.167, Y -14.360, Z 68.000}
   LaserStart_Ext()
   LIN {X 2.357, Y -14.360, Z 68.000}
   LaserEnd_Ext()
   LIN {X -1.080, Y -14.360, Z 68.000}
   LaserStart_Ext()
   LIN {X -5.892, Y -14.360, Z 68.000}
   LaserEnd_Ext()
   LIN {X -5.534, Y -13.360, Z 68.000}
   LaserStart_Ext()
   LIN {X 9.244, Y -13.360, Z 68.000}
   LaserEnd_Ext()
   LIN {X 9.321, Y -12.360, Z 68.000}
   LaserStart_Ext()
   LIN {X -5.186, Y -12.360, Z 68.000}
   LaserEnd_Ext()
   LIN {X -4.838, Y -11.360, Z 68.000}
   LaserStart_Ext()
   LIN {X 9.399, Y -11.360, Z 68.000}
   LaserEnd_Ext()
   LIN {X 9.439, Y -10.360, Z 68.000}
   LaserStart_Ext()
   LIN {X -4.493, Y -10.360, Z 68.000}
   LaserEnd_Ext()
   LIN {X -4.200, Y -9.360, Z 68.000}
   LaserStart_Ext()
   LIN {X 9.477, Y -9.360, Z 68.000}
   LaserEnd_Ext()
   LIN {X 9.516, Y -8.360, Z 68.000}
   LaserStart_Ext()
   LIN {X -3.911, Y -8.360, Z 68.000}
   LaserEnd_Ext()
   LIN {X -3.622, Y -7.360, Z 68.000}
   LaserStart_Ext()
   LIN {X 9.554, Y -7.360, Z 68.000}
   LaserEnd_Ext()
   LIN {X 9.581, Y -6.360, Z 68.000}
   LaserStart_Ext()
   LIN {X -3.359, Y -6.360, Z 68.000}
   LaserEnd_Ext()
   LIN {X -3.140, Y -5.360, Z 68.000}
   LaserStart_Ext()
   LIN {X 9.572, Y -5.360, Z 68.000}
   LaserEnd_Ext()
   LIN {X 9.563, Y -4.360, Z 68.000}
   LaserStart_Ext()
   LIN {X -2.921, Y -4.360, Z 68.000}
   LaserEnd_Ext()
   LIN {X -2.702, Y -3.360, Z 68.000}
   LaserStart_Ext()
   LIN {X 9.552, Y -3.360, Z 68.000}
   LaserEnd_Ext()
   LIN {X 9.536, Y -2.360, Z 68.000}
   LaserStart_Ext()
   LIN {X -2.483, Y -2.360, Z 68.000}
   LaserEnd_Ext()
   LIN {X -2.262, Y -1.360, Z 68.000}
   LaserStart_Ext()
   LIN {X 9.520, Y -1.360, Z 68.000}
   LaserEnd_Ext()
   LIN {X 9.504, Y -0.360, Z 68.000}
   LaserStart_Ext()
   LIN {X -2.086, Y -0.360, Z 68.000}
   LaserEnd_Ext()
   LIN {X -1.943, Y 0.640, Z 68.000}
   LaserStart_Ext()
   LIN {X 9.453, Y 0.640, Z 68.000}
   LaserEnd_Ext()
   LIN {X 9.392, Y 1.640, Z 68.000}
   LaserStart_Ext()
   LIN {X -1.808, Y 1.640, Z 68.000}
   LaserEnd_Ext()
   LIN {X -1.673, Y 2.640, Z 68.000}
   LaserStart_Ext()
   LIN {X 9.330, Y 2.640, Z 68.000}
   LaserEnd_Ext()
   LIN {X 9.269, Y 3.640, Z 68.000}
   LaserStart_Ext()
   LIN {X -1.538, Y 3.640, Z 68.000}
   LaserEnd_Ext()
   LIN {X -1.403, Y 4.640, Z 68.000}
   LaserStart_Ext()
   LIN {X 9.207, Y 4.640, Z 68.000}
   LaserEnd_Ext()
   LIN {X 9.100, Y 5.640, Z 68.000}
   LaserStart_Ext()
   LIN {X -1.328, Y 5.640, Z 68.000}
   LaserEnd_Ext()
   LIN {X -1.290, Y 6.640, Z 68.000}
   LaserStart_Ext()
   LIN {X 8.987, Y 6.640, Z 68.000}
   LaserEnd_Ext()
   LIN {X 8.857, Y 7.640, Z 68.000}
   LaserStart_Ext()
   LIN {X -1.251, Y 7.640, Z 68.000}
   LaserEnd_Ext()
   LIN {X -1.223, Y 8.640, Z 68.000}
   LaserStart_Ext()
   LIN {X 8.701, Y 8.640, Z 68.000}
   LaserEnd_Ext()
   LIN {X 8.546, Y 9.640, Z 68.000}
   LaserStart_Ext()
   LIN {X -1.215, Y 9.640, Z 68.000}
   LaserEnd_Ext()
   LIN {X -1.207, Y 10.640, Z 68.000}
   LaserStart_Ext()
   LIN {X 8.390, Y 10.640, Z 68.000}
   LaserEnd_Ext()
   LIN {X 8.234, Y 11.640, Z 68.000}
   LaserStart_Ext()
   LIN {X -1.199, Y 11.640, Z 68.000}
   LaserEnd_Ext()
   LIN {X -1.190, Y 12.640, Z 68.000}
   LaserStart_Ext()
   LIN {X 8.079, Y 12.640, Z 68.000}
   LaserEnd_Ext()
   LIN {X 7.923, Y 13.640, Z 68.000}
   LaserStart_Ext()
   LIN {X -1.182, Y 13.640, Z 68.000}
   LaserEnd_Ext()
   LIN {X -1.174, Y 14.640, Z 68.000}
   LaserStart_Ext()
   LIN {X 7.768, Y 14.640, Z 68.000}
   LaserEnd_Ext()
   LIN {X 7.612, Y 15.640, Z 68.000}
   LaserStart_Ext()
   LIN {X -1.166, Y 15.640, Z 68.000}
   LaserEnd_Ext()
   LIN {X -1.265, Y 16.640, Z 68.000}
   LaserStart_Ext()
   LIN {X 7.423, Y 16.640, Z 68.000}
   LaserEnd_Ext()
   LIN {X 7.230, Y 17.640, Z 68.000}
   LaserStart_Ext()
   LIN {X -1.371, Y 17.640, Z 68.000}
   LaserEnd_Ext()
   LIN {X -1.478, Y 18.640, Z 68.000}
   LaserStart_Ext()
   LIN {X 7.037, Y 18.640, Z 68.000}
   LaserEnd_Ext()
   LIN {X 6.813, Y 19.640, Z 68.000}
   LaserStart_Ext()
   LIN {X -1.584, Y 19.640, Z 68.000}
   LaserEnd_Ext()
   LIN {X -1.690, Y 20.640, Z 68.000}
   LaserStart_Ext()
   LIN {X 6.550, Y 20.640, Z 68.000}
   LaserEnd_Ext()
   LIN {X 6.287, Y 21.640, Z 68.000}
   LaserStart_Ext()
   LIN {X -1.796, Y 21.640, Z 68.000}
   LaserEnd_Ext()
   LIN {X -1.903, Y 22.640, Z 68.000}
   LaserStart_Ext()
   LIN {X 6.024, Y 22.640, Z 68.000}
   LaserEnd_Ext()
   LIN {X 5.760, Y 23.640, Z 68.000}
   LaserStart_Ext()
   LIN {X -1.992, Y 23.640, Z 68.000}
   LaserEnd_Ext()
   LIN {X -2.147, Y 24.640, Z 68.000}
   LaserStart_Ext()
   LIN {X 5.505, Y 24.640, Z 68.000}
   LaserEnd_Ext()
   LIN {X 5.252, Y 25.640, Z 68.000}
   LaserStart_Ext()
   LIN {X -2.344, Y 25.640, Z 68.000}
   LaserEnd_Ext()
   LIN {X -2.544, Y 26.640, Z 68.000}
   LaserStart_Ext()
   LIN {X 4.988, Y 26.640, Z 68.000}
   LaserEnd_Ext()
   LIN {X 4.665, Y 27.640, Z 68.000}
   LaserStart_Ext()
   LIN {X -2.743, Y 27.640, Z 68.000}
   LaserEnd_Ext()
   LIN {X -2.943, Y 28.640, Z 68.000}
   LaserStart_Ext()
   LIN {X 4.341, Y 28.640, Z 68.000}
   LaserEnd_Ext()
   LIN {X 4.015, Y 29.640, Z 68.000}
   LaserStart_Ext()
   LIN {X -3.201, Y 29.640, Z 68.000}
   LaserEnd_Ext()
   LIN {X -3.463, Y 30.640, Z 68.000}
   LaserStart_Ext()
   LIN {X 3.690, Y 30.640, Z 68.000}
   LaserEnd_Ext()
   LIN {X 3.361, Y 31.640, Z 68.000}
   LaserStart_Ext()
   LIN {X -3.723, Y 31.640, Z 68.000}
   LaserEnd_Ext()
   LIN {X -3.989, Y 32.640, Z 68.000}
   LaserStart_Ext()
   LIN {X 2.997, Y 32.640, Z 68.000}
   LaserEnd_Ext()
   LIN {X 2.634, Y 33.640, Z 68.000}
   LaserStart_Ext()
   LIN {X -4.298, Y 33.640, Z 68.000}
   LaserEnd_Ext()
   LIN {X -4.609, Y 34.640, Z 68.000}
   LaserStart_Ext()
   LIN {X 2.243, Y 34.640, Z 68.000}
   LaserEnd_Ext()
   LIN {X 1.849, Y 35.640, Z 68.000}
   LaserStart_Ext()
   LIN {X -4.935, Y 35.640, Z 68.000}
   LaserEnd_Ext()
   LIN {X -5.286, Y 36.640, Z 68.000}
   LaserStart_Ext()
   LIN {X 1.456, Y 36.640, Z 68.000}
   LaserEnd_Ext()
   LIN {X 1.044, Y 37.640, Z 68.000}
   LaserStart_Ext()
   LIN {X -5.637, Y 37.640, Z 68.000}
   LaserEnd_Ext()
   LIN {X -6.018, Y 38.640, Z 68.000}
   LaserStart_Ext()
   LIN {X 0.616, Y 38.640, Z 68.000}
   LaserEnd_Ext()
   LIN {X 0.187, Y 39.640, Z 68.000}
   LaserStart_Ext()
   LIN {X -6.408, Y 39.640, Z 68.000}
   LaserEnd_Ext()
   LIN {X -6.724, Y 40.640, Z 68.000}
   LaserStart_Ext()
   LIN {X -0.265, Y 40.640, Z 68.000}
   LaserEnd_Ext()
   LIN {X -0.724, Y 41.640, Z 68.000}
   LaserStart_Ext()
   LIN {X -6.767, Y 41.640, Z 68.000}
   LaserEnd_Ext()
   LIN {X -6.540, Y 42.640, Z 68.000}
   LaserStart_Ext()
   LIN {X -1.216, Y 42.640, Z 68.000}
   LaserEnd_Ext()
   LIN {X -2.081, Y 43.640, Z 68.000}
   LaserStart_Ext()
   LIN {X -5.582, Y 43.640, Z 68.000}
   LaserEnd_Ext()
   LIN {X -3.540, Y -17.108, Z 68.850}
   LaserStart_Ext()
   LIN {X -1.993, Y -15.682, Z 68.850} C_DIS
   LIN {X -0.771, Y -15.279, Z 68.850} C_DIS
   LIN {X -0.016, Y -15.031, Z 68.850} C_DIS
   LIN {X 1.028, Y -15.125, Z 68.850} C_DIS
   LIN {X 2.018, Y -15.217, Z 68.850} C_DIS
   LIN {X 2.727, Y -15.623, Z 68.850} C_DIS
   LIN {X 3.865, Y -16.267, Z 68.850} C_DIS
   LIN {X 4.817, Y -17.714, Z 68.850} C_DIS
   LIN {X 5.261, Y -18.393, Z 68.850} C_DIS
   LIN {X 5.333, Y -19.137, Z 68.850} C_DIS
   LIN {X 5.477, Y -20.592, Z 68.850} C_DIS
   LIN {X 5.162, Y -21.421, Z 68.850} C_DIS
   LIN {X 4.623, Y -22.825, Z 68.850} C_DIS
   LIN {X 3.573, Y -23.827, Z 68.850} C_DIS
   LIN {X 3.112, Y -24.265, Z 68.850} C_DIS
   LIN {X 2.114, Y -24.605, Z 68.850} C_DIS
   LIN {X 1.028, Y -24.978, Z 68.850} C_DIS
   LIN {X 0.334, Y -24.915, Z 68.850} C_DIS
   LIN {X -1.009, Y -24.789, Z 68.850} C_DIS
   LIN {X -2.591, Y -23.896, Z 68.850} C_DIS
   LIN {X -2.809, Y -23.774, Z 68.850} C_DIS
   LIN {X -2.936, Y -23.605, Z 68.850} C_DIS
   LIN {X -4.054, Y -22.104, Z 68.850} C_DIS
   LIN {X -4.442, Y -20.310, Z 68.850} C_DIS
   LIN {X -4.496, Y -20.065, Z 68.850} C_DIS
   LIN {X -3.583, Y -17.165, Z 68.850} C_DIS
   LIN {X -3.540, Y -17.108, Z 68.850}
   LaserEnd_Ext()
   LIN {X 10.631, Y -6.519, Z 68.850}
   LaserStart_Ext()
   LIN {X 10.626, Y -5.911, Z 68.850} C_DIS
   LIN {X 10.532, Y -0.005, Z 68.850} C_DIS
   LIN {X 10.424, Y 1.749, Z 68.850} C_DIS
   LIN {X 10.300, Y 3.753, Z 68.850} C_DIS
   LIN {X 10.251, Y 4.553, Z 68.850} C_DIS
   LIN {X 9.900, Y 7.664, Z 68.850} C_DIS
   LIN {X 8.787, Y 14.818, Z 68.850} C_DIS
   LIN {X 7.864, Y 19.600, Z 68.850} C_DIS
   LIN {X 6.216, Y 25.860, Z 68.850} C_DIS
   LIN {X 5.987, Y 26.763, Z 68.850} C_DIS
   LIN {X 5.782, Y 27.396, Z 68.850} C_DIS
   LIN {X 4.712, Y 30.683, Z 68.850} C_DIS
   LIN {X 4.395, Y 31.656, Z 68.850} C_DIS
   LIN {X 4.276, Y 31.983, Z 68.850} C_DIS
   LIN {X 3.474, Y 34.183, Z 68.850} C_DIS
   LIN {X 2.686, Y 36.180, Z 68.850} C_DIS
   LIN {X 2.147, Y 37.526, Z 68.850} C_DIS
   LIN {X 1.179, Y 39.776, Z 68.850} C_DIS
   LIN {X 1.072, Y 40.027, Z 68.850} C_DIS
   LIN {X 1.027, Y 40.126, Z 68.850} C_DIS
   LIN {X 0.279, Y 41.772, Z 68.850} C_DIS
   LIN {X -0.142, Y 42.663, Z 68.850} C_DIS
   LIN {X -0.355, Y 43.114, Z 68.850} C_DIS
   LIN {X -0.727, Y 43.619, Z 68.850} C_DIS
   LIN {X -1.226, Y 44.300, Z 68.850} C_DIS
   LIN {X -1.880, Y 44.691, Z 68.850} C_DIS
   LIN {X -2.721, Y 45.190, Z 68.850} C_DIS
   LIN {X -4.373, Y 45.352, Z 68.850} C_DIS
   LIN {X -4.494, Y 45.344, Z 68.850} C_DIS
   LIN {X -6.818, Y 44.183, Z 68.850} C_DIS
   LIN {X -7.198, Y 43.620, Z 68.850} C_DIS
   LIN {X -7.712, Y 42.725, Z 68.850} C_DIS
   LIN {X -7.912, Y 41.421, Z 68.850} C_DIS
   LIN {X -7.938, Y 41.272, Z 68.850} C_DIS
   LIN {X -7.913, Y 41.168, Z 68.850} C_DIS
   LIN {X -7.625, Y 39.878, Z 68.850} C_DIS
   LIN {X -7.234, Y 38.896, Z 68.850} C_DIS
   LIN {X -7.162, Y 38.716, Z 68.850} C_DIS
   LIN {X -7.041, Y 38.398, Z 68.850} C_DIS
   LIN {X -6.590, Y 37.222, Z 68.850} C_DIS
   LIN {X -6.212, Y 36.157, Z 68.850} C_DIS
   LIN {X -5.802, Y 34.986, Z 68.850} C_DIS
   LIN {X -5.152, Y 32.900, Z 68.850} C_DIS
   LIN {X -4.935, Y 32.207, Z 68.850} C_DIS
   LIN {X -4.865, Y 31.947, Z 68.850} C_DIS
   LIN {X -3.940, Y 28.415, Z 68.850} C_DIS
   LIN {X -3.042, Y 23.919, Z 68.850} C_DIS
   LIN {X -2.181, Y 15.866, Z 68.850} C_DIS
   LIN {X -2.249, Y 7.556, Z 68.850} C_DIS
   LIN {X -2.349, Y 4.943, Z 68.850} C_DIS
   LIN {X -2.867, Y 1.108, Z 68.850} C_DIS
   LIN {X -3.204, Y -1.174, Z 68.850} C_DIS
   LIN {X -3.771, Y -3.742, Z 68.850} C_DIS
   LIN {X -4.364, Y -6.447, Z 68.850} C_DIS
   LIN {X -5.183, Y -9.281, Z 68.850} C_DIS
   LIN {X -5.493, Y -10.346, Z 68.850} C_DIS
   LIN {X -5.692, Y -10.918, Z 68.850} C_DIS
   LIN {X -6.682, Y -13.767, Z 68.850} C_DIS
   LIN {X -7.753, Y -16.446, Z 68.850} C_DIS
   LIN {X -7.817, Y -16.653, Z 68.850} C_DIS
   LIN {X -8.496, Y -19.627, Z 68.850} C_DIS
   LIN {X -7.982, Y -22.828, Z 68.850} C_DIS
   LIN {X -7.910, Y -23.291, Z 68.850} C_DIS
   LIN {X -7.698, Y -23.621, Z 68.850} C_DIS
   LIN {X -5.861, Y -26.431, Z 68.850} C_DIS
   LIN {X -3.523, Y -28.089, Z 68.850} C_DIS
   LIN {X 0.005, Y -29.005, Z 68.850} C_DIS
   LIN {X 1.274, Y -28.820, Z 68.850} C_DIS
   LIN {X 3.216, Y -28.585, Z 68.850} C_DIS
   LIN {X 6.243, Y -26.866, Z 68.850} C_DIS
   LIN {X 6.448, Y -26.746, Z 68.850} C_DIS
   LIN {X 6.629, Y -26.509, Z 68.850} C_DIS
   LIN {X 8.514, Y -24.095, Z 68.850} C_DIS
   LIN {X 9.070, Y -22.396, Z 68.850} C_DIS
   LIN {X 9.429, Y -21.279, Z 68.850} C_DIS
   LIN {X 9.720, Y -19.087, Z 68.850} C_DIS
   LIN {X 9.862, Y -18.044, Z 68.850} C_DIS
   LIN {X 9.924, Y -17.480, Z 68.850} C_DIS
   LIN {X 10.174, Y -15.099, Z 68.850} C_DIS
   LIN {X 10.377, Y -12.476, Z 68.850} C_DIS
   LIN {X 10.459, Y -11.304, Z 68.850} C_DIS
   LIN {X 10.589, Y -7.619, Z 68.850} C_DIS
   LIN {X 10.631, Y -6.519, Z 68.850}
   LaserEnd_Ext()
   LIN {X 9.602, Y -7.262, Z 68.850}
   LaserStart_Ext()
   LIN {X 9.602, Y -4.432, Z 68.850}
   LaserEnd_Ext()
   LIN {X 8.602, Y 9.502, Z 68.850}
   LaserStart_Ext()
   LIN {X 8.602, Y -19.912, Z 68.850}
   LaserEnd_Ext()
   LIN {X 7.602, Y -23.639, Z 68.850}
   LaserStart_Ext()
   LIN {X 7.602, Y 15.680, Z 68.850}
   LaserEnd_Ext()
   LIN {X 6.602, Y 20.465, Z 68.850}
   LaserStart_Ext()
   LIN {X 6.602, Y -24.919, Z 68.850}
   LaserEnd_Ext()
   LIN {X 5.602, Y -26.080, Z 68.850}
   LaserStart_Ext()
   LIN {X 5.602, Y -23.066, Z 68.850}
   LaserEnd_Ext()
   LIN {X 5.602, Y -17.087, Z 68.850}
   LaserStart_Ext()
   LIN {X 5.602, Y 24.263, Z 68.850}
   LaserEnd_Ext()
   LIN {X 4.602, Y 27.791, Z 68.850}
   LaserStart_Ext()
   LIN {X 4.602, Y -15.593, Z 68.850}
   LaserEnd_Ext()
   LIN {X 4.602, Y -24.228, Z 68.850}
   LaserStart_Ext()
   LIN {X 4.602, Y -26.648, Z 68.850}
   LaserEnd_Ext()
   LIN {X 3.602, Y -27.216, Z 68.850}
   LaserStart_Ext()
   LIN {X 3.602, Y -25.135, Z 68.850}
   LaserEnd_Ext()
   LIN {X 3.602, Y -14.969, Z 68.850}
   LaserStart_Ext()
   LIN {X 3.602, Y 30.862, Z 68.850}
   LaserEnd_Ext()
   LIN {X 2.602, Y 33.655, Z 68.850}
   LaserStart_Ext()
   LIN {X 2.602, Y -14.399, Z 68.850}
   LaserEnd_Ext()
   LIN {X 2.602, Y -25.495, Z 68.850}
   LaserStart_Ext()
   LIN {X 2.602, Y -27.652, Z 68.850}
   LaserEnd_Ext()
   LIN {X 1.602, Y -27.773, Z 68.850}
   LaserStart_Ext()
   LIN {X 1.602, Y -25.838, Z 68.850}
   LaserEnd_Ext()
   LIN {X 1.602, Y -14.174, Z 68.850}
   LaserStart_Ext()
   LIN {X 1.602, Y 36.196, Z 68.850}
   LaserEnd_Ext()
   LIN {X 0.602, Y 38.588, Z 68.850}
   LaserStart_Ext()
   LIN {X 0.602, Y -14.082, Z 68.850}
   LaserEnd_Ext()
   LIN {X 0.602, Y -25.943, Z 68.850}
   LaserStart_Ext()
   LIN {X 0.602, Y -27.908, Z 68.850}
   LaserEnd_Ext()
   LIN {X -0.398, Y -27.870, Z 68.850}
   LaserStart_Ext()
   LIN {X -0.398, Y -25.851, Z 68.850}
   LaserEnd_Ext()
   LIN {X -0.398, Y -14.104, Z 68.850}
   LaserStart_Ext()
   LIN {X -0.398, Y 40.845, Z 68.850}
   LaserEnd_Ext()
   LIN {X -1.398, Y 42.843, Z 68.850}
   LaserStart_Ext()
   LIN {X -1.398, Y 17.967, Z 68.850}
   LaserEnd_Ext()
   LIN {X -1.398, Y 4.514, Z 68.850}
   LaserStart_Ext()
   LIN {X -1.398, Y -14.433, Z 68.850}
   LaserEnd_Ext()
   LIN {X -1.398, Y -25.710, Z 68.850}
   LaserStart_Ext()
   LIN {X -1.398, Y -27.615, Z 68.850}
   LaserEnd_Ext()
   LIN {X -2.398, Y -27.359, Z 68.850}
   LaserStart_Ext()
   LIN {X -2.398, Y -25.153, Z 68.850}
   LaserEnd_Ext()
   LIN {X -2.398, Y -14.768, Z 68.850}
   LaserStart_Ext()
   LIN {X -2.398, Y -2.161, Z 68.850}
   LaserEnd_Ext()
   LIN {X -2.398, Y 25.800, Z 68.850}
   LaserStart_Ext()
   LIN {X -2.398, Y 43.836, Z 68.850}
   LaserEnd_Ext()
   LIN {X -3.398, Y 44.251, Z 68.850}
   LaserStart_Ext()
   LIN {X -3.398, Y 30.292, Z 68.850}
   LaserEnd_Ext()
   LIN {X -3.398, Y -6.706, Z 68.850}
   LaserStart_Ext()
   LIN {X -3.398, Y -15.617, Z 68.850}
   LaserEnd_Ext()
   LIN {X -3.398, Y -24.582, Z 68.850}
   LaserStart_Ext()
   LIN {X -3.398, Y -26.952, Z 68.850}
   LaserEnd_Ext()
   LIN {X -4.398, Y -26.242, Z 68.850}
   LaserStart_Ext()
   LIN {X -4.398, Y -23.316, Z 68.850}
   LaserEnd_Ext()
   LIN {X -4.398, Y -16.573, Z 68.850}
   LaserStart_Ext()
   LIN {X -4.398, Y -10.162, Z 68.850}
   LaserEnd_Ext()
   LIN {X -4.398, Y 33.842, Z 68.850}
   LaserStart_Ext()
   LIN {X -4.398, Y 44.274, Z 68.850}
   LaserEnd_Ext()
   LIN {X -5.398, Y 43.774, Z 68.850}
   LaserStart_Ext()
   LIN {X -5.398, Y 36.853, Z 68.850}
   LaserEnd_Ext()
   LIN {X -5.398, Y -13.118, Z 68.850}
   LaserStart_Ext()
   LIN {X -5.398, Y -19.600, Z 68.850}
   LaserEnd_Ext()
   LIN {X -5.398, Y -20.620, Z 68.850}
   LaserStart_Ext()
   LIN {X -5.398, Y -25.311, Z 68.850}
   LaserEnd_Ext()
   LIN {X -6.398, Y -23.781, Z 68.850}
   LaserStart_Ext()
   LIN {X -6.398, Y -15.751, Z 68.850}
   LaserEnd_Ext()
   LIN {X -6.398, Y 39.501, Z 68.850}
   LaserStart_Ext()
   LIN {X -6.398, Y 43.006, Z 68.850}
   LaserEnd_Ext()
   LIN {X -7.398, Y -19.311, Z 68.850}
   LaserStart_Ext()
   LIN {X -7.398, Y -20.158, Z 68.850}
   LaserEnd_Ext()
   LIN {X 1.583, Y -15.116, Z 69.700}
   LaserStart_Ext()
   LIN {X 2.086, Y -15.159, Z 69.700} C_DIS
   LIN {X 2.664, Y -15.485, Z 69.700} C_DIS
   LIN {X 3.935, Y -16.206, Z 69.700} C_DIS
   LIN {X 4.793, Y -17.508, Z 69.700} C_DIS
   LIN {X 5.337, Y -18.328, Z 69.700} C_DIS
   LIN {X 5.413, Y -19.069, Z 69.700} C_DIS
   LIN {X 5.557, Y -20.527, Z 69.700} C_DIS
   LIN {X 4.889, Y -22.287, Z 69.700} C_DIS
   LIN {X 4.705, Y -22.767, Z 69.700} C_DIS
   LIN {X 3.938, Y -23.500, Z 69.700} C_DIS
   LIN {X 3.204, Y -24.203, Z 69.700} C_DIS
   LIN {X 2.575, Y -24.423, Z 69.700} C_DIS
   LIN {X 1.119, Y -24.923, Z 69.700} C_DIS
   LIN {X -0.859, Y -24.745, Z 69.700} C_DIS
   LIN {X -0.990, Y -24.699, Z 69.700} C_DIS
   LIN {X -2.721, Y -23.728, Z 69.700} C_DIS
   LIN {X -3.726, Y -22.389, Z 69.700} C_DIS
   LIN {X -3.970, Y -22.061, Z 69.700} C_DIS
   LIN {X -4.055, Y -21.670, Z 69.700} C_DIS
   LIN {X -4.417, Y -20.023, Z 69.700} C_DIS
   LIN {X -3.846, Y -18.212, Z 69.700} C_DIS
   LIN {X -3.515, Y -17.114, Z 69.700} C_DIS
   LIN {X -1.914, Y -15.635, Z 69.700} C_DIS
   LIN {X 0.051, Y -14.979, Z 69.700} C_DIS
   LIN {X 1.583, Y -15.116, Z 69.700}
   LaserEnd_Ext()
   LIN {X -3.320, Y 25.201, Z 69.700}
   LaserStart_Ext()
   LIN {X -3.949, Y 28.350, Z 69.700} C_DIS
   LIN {X -4.597, Y 30.823, Z 69.700} C_DIS
   LIN {X -4.978, Y 32.248, Z 69.700} C_DIS
   LIN {X -5.536, Y 34.025, Z 69.700} C_DIS
   LIN {X -5.852, Y 35.025, Z 69.700} C_DIS
   LIN {X -6.130, Y 35.805, Z 69.700} C_DIS
   LIN {X -6.645, Y 37.259, Z 69.700} C_DIS
   LIN {X -6.886, Y 37.888, Z 69.700} C_DIS
   LIN {X -7.221, Y 38.751, Z 69.700} C_DIS
   LIN {X -7.655, Y 39.835, Z 69.700} C_DIS
   LIN {X -7.719, Y 40.074, Z 69.700} C_DIS
   LIN {X -8.004, Y 41.407, Z 69.700} C_DIS
   LIN {X -7.871, Y 42.463, Z 69.700} C_DIS
   LIN {X -7.834, Y 42.574, Z 69.700} C_DIS
   LIN {X -6.946, Y 44.159, Z 69.700} C_DIS
   LIN {X -6.853, Y 44.248, Z 69.700} C_DIS
   LIN {X -6.409, Y 44.447, Z 69.700} C_DIS
   LIN {X -4.532, Y 45.402, Z 69.700} C_DIS
   LIN {X -3.213, Y 45.277, Z 69.700} C_DIS
   LIN {X -2.794, Y 45.235, Z 69.700} C_DIS
   LIN {X -2.207, Y 44.887, Z 69.700} C_DIS
   LIN {X -1.297, Y 44.349, Z 69.700} C_DIS
   LIN {X -0.919, Y 43.838, Z 69.700} C_DIS
   LIN {X -0.424, Y 43.165, Z 69.700} C_DIS
   LIN {X 0.041, Y 42.184, Z 69.700} C_DIS
   LIN {X 0.213, Y 41.825, Z 69.700} C_DIS
   LIN {X 0.366, Y 41.492, Z 69.700} C_DIS
   LIN {X 1.011, Y 40.082, Z 69.700} C_DIS
   LIN {X 1.303, Y 39.418, Z 69.700} C_DIS
   LIN {X 2.054, Y 37.671, Z 69.700} C_DIS
   LIN {X 3.403, Y 34.300, Z 69.700} C_DIS
   LIN {X 3.442, Y 34.199, Z 69.700} C_DIS
   LIN {X 4.457, Y 31.425, Z 69.700} C_DIS
   LIN {X 5.776, Y 27.371, Z 69.700} C_DIS
   LIN {X 6.045, Y 26.529, Z 69.700} C_DIS
   LIN {X 7.826, Y 19.766, Z 69.700} C_DIS
   LIN {X 8.991, Y 13.730, Z 69.700} C_DIS
   LIN {X 9.889, Y 7.959, Z 69.700} C_DIS
   LIN {X 10.306, Y 4.268, Z 69.700} C_DIS
   LIN {X 10.364, Y 3.320, Z 69.700} C_DIS
   LIN {X 10.510, Y 0.943, Z 69.700} C_DIS
   LIN {X 10.564, Y 0.073, Z 69.700} C_DIS
   LIN {X 10.623, Y -3.673, Z 69.700} C_DIS
   LIN {X 10.678, Y -6.442, Z 69.700} C_DIS
   LIN {X 10.644, Y -7.637, Z 69.700} C_DIS
   LIN {X 10.518, Y -11.227, Z 69.700} C_DIS
   LIN {X 10.345, Y -13.682, Z 69.700} C_DIS
   LIN {X 10.242, Y -15.023, Z 69.700} C_DIS
   LIN {X 10.039, Y -16.956, Z 69.700} C_DIS
   LIN {X 9.937, Y -17.968, Z 69.700} C_DIS
   LIN {X 9.854, Y -18.626, Z 69.700} C_DIS
   LIN {X 9.511, Y -21.204, Z 69.700} C_DIS
   LIN {X 8.776, Y -23.496, Z 69.700} C_DIS
   LIN {X 8.603, Y -24.023, Z 69.700} C_DIS
   LIN {X 8.019, Y -24.771, Z 69.700} C_DIS
   LIN {X 6.618, Y -26.608, Z 69.700} C_DIS
   LIN {X 5.038, Y -27.533, Z 69.700} C_DIS
   LIN {X 3.258, Y -28.543, Z 69.700} C_DIS
   LIN {X 0.219, Y -28.912, Z 69.700} C_DIS
   LIN {X -0.032, Y -28.948, Z 69.700} C_DIS
   LIN {X -0.739, Y -28.768, Z 69.700} C_DIS
   LIN {X -3.461, Y -28.034, Z 69.700} C_DIS
   LIN {X -4.224, Y -27.487, Z 69.700} C_DIS
   LIN {X -5.766, Y -26.392, Z 69.700} C_DIS
   LIN {X -7.229, Y -24.155, Z 69.700} C_DIS
   LIN {X -7.823, Y -23.258, Z 69.700} C_DIS
   LIN {X -8.062, Y -21.814, Z 69.700} C_DIS
   LIN {X -8.418, Y -19.595, Z 69.700} C_DIS
   LIN {X -8.032, Y -17.906, Z 69.700} C_DIS
   LIN {X -7.719, Y -16.503, Z 69.700} C_DIS
   LIN {X -7.141, Y -15.040, Z 69.700} C_DIS
   LIN {X -6.616, Y -13.725, Z 69.700} C_DIS
   LIN {X -6.164, Y -12.426, Z 69.700} C_DIS
   LIN {X -5.566, Y -10.706, Z 69.700} C_DIS
   LIN {X -4.634, Y -7.504, Z 69.700} C_DIS
   LIN {X -4.316, Y -6.404, Z 69.700} C_DIS
   LIN {X -4.086, Y -5.353, Z 69.700} C_DIS
   LIN {X -3.248, Y -1.554, Z 69.700} C_DIS
   LIN {X -2.749, Y 1.823, Z 69.700} C_DIS
   LIN {X -2.349, Y 4.782, Z 69.700} C_DIS
   LIN {X -2.271, Y 6.797, Z 69.700} C_DIS
   LIN {X -2.195, Y 16.082, Z 69.700} C_DIS
   LIN {X -2.946, Y 23.146, Z 69.700} C_DIS
   LIN {X -3.093, Y 24.118, Z 69.700} C_DIS
   LIN {X -3.320, Y 25.201, Z 69.700}
   LaserEnd_Ext()
   LIN {X -6.028, Y 43.522, Z 69.700}
   LaserStart_Ext()
   LIN {X -1.929, Y 43.522, Z 69.700}
   LaserEnd_Ext()
   LIN {X -1.226, Y 42.522, Z 69.700}
   LaserStart_Ext()
   LIN {X -6.717, Y 42.522, Z 69.700}
   LaserEnd_Ext()
   LIN {X -6.982, Y 41.522, Z 69.700}
   LaserStart_Ext()
   LIN {X -0.750, Y 41.522, Z 69.700}
   LaserEnd_Ext()
   LIN {X -0.290, Y 40.522, Z 69.700}
   LaserStart_Ext()
   LIN {X -6.792, Y 40.522, Z 69.700}
   LaserEnd_Ext()
   LIN {X -6.452, Y 39.522, Z 69.700}
   LaserStart_Ext()
   LIN {X 0.165, Y 39.522, Z 69.700}
   LaserEnd_Ext()
   LIN {X 0.600, Y 38.522, Z 69.700}
   LaserStart_Ext()
   LIN {X -6.059, Y 38.522, Z 69.700}
   LaserEnd_Ext()
   LIN {X -5.677, Y 37.522, Z 69.700}
   LaserStart_Ext()
   LIN {X 1.030, Y 37.522, Z 69.700}
   LaserEnd_Ext()
   LIN {X 1.437, Y 36.522, Z 69.700}
   LaserStart_Ext()
   LIN {X -5.323, Y 36.522, Z 69.700}
   LaserEnd_Ext()
   LIN {X -4.967, Y 35.522, Z 69.700}
   LaserStart_Ext()
   LIN {X 1.837, Y 35.522, Z 69.700}
   LaserEnd_Ext()
   LIN {X 2.237, Y 34.522, Z 69.700}
   LaserStart_Ext()
   LIN {X -4.644, Y 34.522, Z 69.700}
   LaserEnd_Ext()
   LIN {X -4.330, Y 33.522, Z 69.700}
   LaserStart_Ext()
   LIN {X 2.625, Y 33.522, Z 69.700}
   LaserEnd_Ext()
   LIN {X 2.991, Y 32.522, Z 69.700}
   LaserStart_Ext()
   LIN {X -4.016, Y 32.522, Z 69.700}
   LaserEnd_Ext()
   LIN {X -3.749, Y 31.522, Z 69.700}
   LaserStart_Ext()
   LIN {X 3.357, Y 31.522, Z 69.700}
   LaserEnd_Ext()
   LIN {X 3.699, Y 30.522, Z 69.700}
   LaserStart_Ext()
   LIN {X -3.484, Y 30.522, Z 69.700}
   LaserEnd_Ext()
   LIN {X -3.223, Y 29.522, Z 69.700}
   LaserStart_Ext()
   LIN {X 4.025, Y 29.522, Z 69.700}
   LaserEnd_Ext()
   LIN {X 4.350, Y 28.522, Z 69.700}
   LaserStart_Ext()
   LIN {X -2.964, Y 28.522, Z 69.700}
   LaserEnd_Ext()
   LIN {X -2.764, Y 27.522, Z 69.700}
   LaserStart_Ext()
   LIN {X 4.675, Y 27.522, Z 69.700}
   LaserEnd_Ext()
   LIN {X 4.998, Y 26.522, Z 69.700}
   LaserStart_Ext()
   LIN {X -2.564, Y 26.522, Z 69.700}
   LaserEnd_Ext()
   LIN {X -2.365, Y 25.522, Z 69.700}
   LaserStart_Ext()
   LIN {X 5.276, Y 25.522, Z 69.700}
   LaserEnd_Ext()
   LIN {X 5.540, Y 24.522, Z 69.700}
   LaserStart_Ext()
   LIN {X -2.156, Y 24.522, Z 69.700}
   LaserEnd_Ext()
   LIN {X -1.991, Y 23.522, Z 69.700}
   LaserStart_Ext()
   LIN {X 5.803, Y 23.522, Z 69.700}
   LaserEnd_Ext()
   LIN {X 6.066, Y 22.522, Z 69.700}
   LaserStart_Ext()
   LIN {X -1.874, Y 22.522, Z 69.700}
   LaserEnd_Ext()
   LIN {X -1.767, Y 21.522, Z 69.700}
   LaserStart_Ext()
   LIN {X 6.330, Y 21.522, Z 69.700}
   LaserEnd_Ext()
   LIN {X 6.593, Y 20.522, Z 69.700}
   LaserStart_Ext()
   LIN {X -1.661, Y 20.522, Z 69.700}
   LaserEnd_Ext()
   LIN {X -1.555, Y 19.522, Z 69.700}
   LaserStart_Ext()
   LIN {X 6.855, Y 19.522, Z 69.700}
   LaserEnd_Ext()
   LIN {X 7.048, Y 18.522, Z 69.700}
   LaserStart_Ext()
   LIN {X -1.449, Y 18.522, Z 69.700}
   LaserEnd_Ext()
   LIN {X -1.343, Y 17.522, Z 69.700}
   LaserStart_Ext()
   LIN {X 7.241, Y 17.522, Z 69.700}
   LaserEnd_Ext()
   LIN {X 7.434, Y 16.522, Z 69.700}
   LaserStart_Ext()
   LIN {X -1.236, Y 16.522, Z 69.700}
   LaserEnd_Ext()
   LIN {X -1.200, Y 15.522, Z 69.700}
   LaserStart_Ext()
   LIN {X 7.627, Y 15.522, Z 69.700}
   LaserEnd_Ext()
   LIN {X 7.820, Y 14.522, Z 69.700}
   LaserStart_Ext()
   LIN {X -1.208, Y 14.522, Z 69.700}
   LaserEnd_Ext()
   LIN {X -1.216, Y 13.522, Z 69.700}
   LaserStart_Ext()
   LIN {X 8.011, Y 13.522, Z 69.700}
   LaserEnd_Ext()
   LIN {X 8.167, Y 12.522, Z 69.700}
   LaserStart_Ext()
   LIN {X -1.224, Y 12.522, Z 69.700}
   LaserEnd_Ext()
   LIN {X -1.233, Y 11.522, Z 69.700}
   LaserStart_Ext()
   LIN {X 8.322, Y 11.522, Z 69.700}
   LaserEnd_Ext()
   LIN {X 8.478, Y 10.522, Z 69.700}
   LaserStart_Ext()
   LIN {X -1.241, Y 10.522, Z 69.700}
   LaserEnd_Ext()
   LIN {X -1.249, Y 9.522, Z 69.700}
   LaserStart_Ext()
   LIN {X 8.634, Y 9.522, Z 69.700}
   LaserEnd_Ext()
   LIN {X 8.789, Y 8.522, Z 69.700}
   LaserStart_Ext()
   LIN {X -1.257, Y 8.522, Z 69.700}
   LaserEnd_Ext()
   LIN {X -1.265, Y 7.522, Z 69.700}
   LaserStart_Ext()
   LIN {X 8.932, Y 7.522, Z 69.700}
   LaserEnd_Ext()
   LIN {X 9.045, Y 6.522, Z 69.700}
   LaserStart_Ext()
   LIN {X -1.281, Y 6.522, Z 69.700}
   LaserEnd_Ext()
   LIN {X -1.320, Y 5.522, Z 69.700}
   LaserStart_Ext()
   LIN {X 9.158, Y 5.522, Z 69.700}
   LaserEnd_Ext()
   LIN {X 9.271, Y 4.522, Z 69.700}
   LaserStart_Ext()
   LIN {X -1.375, Y 4.522, Z 69.700}
   LaserEnd_Ext()
   LIN {X -1.510, Y 3.522, Z 69.700}
   LaserStart_Ext()
   LIN {X 9.350, Y 3.522, Z 69.700}
   LaserEnd_Ext()
   LIN {X 9.411, Y 2.522, Z 69.700}
   LaserStart_Ext()
   LIN {X -1.645, Y 2.522, Z 69.700}
   LaserEnd_Ext()
   LIN {X -1.782, Y 1.522, Z 69.700}
   LaserStart_Ext()
   LIN {X 9.473, Y 1.522, Z 69.700}
   LaserEnd_Ext()
   LIN {X 9.534, Y 0.522, Z 69.700}
   LaserStart_Ext()
   LIN {X -1.930, Y 0.522, Z 69.700}
   LaserEnd_Ext()
   LIN {X -2.078, Y -0.478, Z 69.700}
   LaserStart_Ext()
   LIN {X 9.573, Y -0.478, Z 69.700}
   LaserEnd_Ext()
   LIN {X 9.588, Y -1.478, Z 69.700}
   LaserStart_Ext()
   LIN {X -2.226, Y -1.478, Z 69.700}
   LaserEnd_Ext()
   LIN {X -2.428, Y -2.478, Z 69.700}
   LaserStart_Ext()
   LIN {X 9.604, Y -2.478, Z 69.700}
   LaserEnd_Ext()
   LIN {X 9.620, Y -3.478, Z 69.700}
   LaserStart_Ext()
   LIN {X -2.648, Y -3.478, Z 69.700}
   LaserEnd_Ext()
   LIN {X -2.869, Y -4.478, Z 69.700}
   LaserStart_Ext()
   LIN {X 9.639, Y -4.478, Z 69.700}
   LaserEnd_Ext()
   LIN {X 9.659, Y -5.478, Z 69.700}
   LaserStart_Ext()
   LIN {X -3.090, Y -5.478, Z 69.700}
   LaserEnd_Ext()
   LIN {X -3.309, Y -6.478, Z 69.700}
   LaserStart_Ext()
   LIN {X 9.677, Y -6.478, Z 69.700}
   LaserEnd_Ext()
   LIN {X 9.649, Y -7.478, Z 69.700}
   LaserStart_Ext()
   LIN {X -3.586, Y -7.478, Z 69.700}
   LaserEnd_Ext()
   LIN {X -3.876, Y -8.478, Z 69.700}
   LaserStart_Ext()
   LIN {X 9.614, Y -8.478, Z 69.700}
   LaserEnd_Ext()
   LIN {X 9.579, Y -9.478, Z 69.700}
   LaserStart_Ext()
   LIN {X -4.167, Y -9.478, Z 69.700}
   LaserEnd_Ext()
   LIN {X -4.458, Y -10.478, Z 69.700}
   LaserStart_Ext()
   LIN {X 9.543, Y -10.478, Z 69.700}
   LaserEnd_Ext()
   LIN {X 9.498, Y -11.478, Z 69.700}
   LaserStart_Ext()
   LIN {X -4.776, Y -11.478, Z 69.700}
   LaserEnd_Ext()
   LIN {X -5.124, Y -12.478, Z 69.700}
   LaserStart_Ext()
   LIN {X 9.427, Y -12.478, Z 69.700}
   LaserEnd_Ext()
   LIN {X 9.357, Y -13.478, Z 69.700}
   LaserStart_Ext()
   LIN {X -5.471, Y -13.478, Z 69.700}
   LaserEnd_Ext()
   LIN {X -5.840, Y -14.478, Z 69.700}
   LaserStart_Ext()
   LIN {X -1.630, Y -14.478, Z 69.700}
   LaserEnd_Ext()
   LIN {X 2.914, Y -14.478, Z 69.700}
   LaserStart_Ext()
   LIN {X 9.281, Y -14.478, Z 69.700}
   LaserEnd_Ext()
   LIN {X 9.189, Y -15.478, Z 69.700}
   LaserStart_Ext()
   LIN {X 4.619, Y -15.478, Z 69.700}
   LaserEnd_Ext()
   LIN {X -3.218, Y -15.478, Z 69.700}
   LaserStart_Ext()
   LIN {X -6.239, Y -15.478, Z 69.700}
   LaserEnd_Ext()
   LIN {X -6.634, Y -16.478, Z 69.700}
   LaserStart_Ext()
   LIN {X -4.286, Y -16.478, Z 69.700}
   LaserEnd_Ext()
   LIN {X 5.312, Y -16.478, Z 69.700}
   LaserStart_Ext()
   LIN {X 9.084, Y -16.478, Z 69.700}
   LaserEnd_Ext()
   LIN {X 8.981, Y -17.478, Z 69.700}
   LaserStart_Ext()
   LIN {X 5.973, Y -17.478, Z 69.700}
   LaserEnd_Ext()
   LIN {X -4.670, Y -17.478, Z 69.700}
   LaserStart_Ext()
   LIN {X -6.912, Y -17.478, Z 69.700}
   LaserEnd_Ext()
   LIN {X -7.137, Y -18.478, Z 69.700}
   LaserStart_Ext()
   LIN {X -4.979, Y -18.478, Z 69.700}
   LaserEnd_Ext()
   LIN {X 6.358, Y -18.478, Z 69.700}
   LaserStart_Ext()
   LIN {X 8.864, Y -18.478, Z 69.700}
   LaserEnd_Ext()
   LIN {X 8.732, Y -19.478, Z 69.700}
   LaserStart_Ext()
   LIN {X 6.458, Y -19.478, Z 69.700}
   LaserEnd_Ext()
   LIN {X -5.294, Y -19.478, Z 69.700}
   LaserStart_Ext()
   LIN {X -7.366, Y -19.478, Z 69.700}
   LaserEnd_Ext()
   LIN {X -7.263, Y -20.478, Z 69.700}
   LaserStart_Ext()
   LIN {X -5.340, Y -20.478, Z 69.700}
   LaserEnd_Ext()
   LIN {X 6.555, Y -20.478, Z 69.700}
   LaserStart_Ext()
   LIN {X 8.599, Y -20.478, Z 69.700}
   LaserEnd_Ext()
   LIN {X 8.373, Y -21.478, Z 69.700}
   LaserStart_Ext()
   LIN {X 6.266, Y -21.478, Z 69.700}
   LaserEnd_Ext()
   LIN {X -5.121, Y -21.478, Z 69.700}
   LaserStart_Ext()
   LIN {X -7.103, Y -21.478, Z 69.700}
   LaserEnd_Ext()
   LIN {X -6.938, Y -22.478, Z 69.700}
   LaserStart_Ext()
   LIN {X -4.878, Y -22.478, Z 69.700}
   LaserEnd_Ext()
   LIN {X 5.886, Y -22.478, Z 69.700}
   LaserStart_Ext()
   LIN {X 8.052, Y -22.478, Z 69.700}
   LaserEnd_Ext()
   LIN {X 7.729, Y -23.478, Z 69.700}
   LaserStart_Ext()
   LIN {X 5.407, Y -23.478, Z 69.700}
   LaserEnd_Ext()
   LIN {X -4.159, Y -23.478, Z 69.700}
   LaserStart_Ext()
   LIN {X -6.478, Y -23.478, Z 69.700}
   LaserEnd_Ext()
   LIN {X -5.823, Y -24.478, Z 69.700}
   LaserStart_Ext()
   LIN {X -3.382, Y -24.478, Z 69.700}
   LaserEnd_Ext()
   LIN {X 4.362, Y -24.478, Z 69.700}
   LaserStart_Ext()
   LIN {X 6.984, Y -24.478, Z 69.700}
   LaserEnd_Ext()
   LIN {X 6.222, Y -25.478, Z 69.700}
   LaserStart_Ext()
   LIN {X 2.580, Y -25.478, Z 69.700}
   LaserEnd_Ext()
   LIN {X -1.645, Y -25.478, Z 69.700}
   LaserStart_Ext()
   LIN {X -5.169, Y -25.478, Z 69.700}
   LaserEnd_Ext()
   LIN {X -3.917, Y -26.478, Z 69.700}
   LaserStart_Ext()
   LIN {X 4.860, Y -26.478, Z 69.700}
   LaserEnd_Ext()
   LIN {X 3.108, Y -27.478, Z 69.700}
   LaserStart_Ext()
   LIN {X -1.679, Y -27.478, Z 69.700}
   LaserEnd_Ext()
   LIN {X -1.963, Y -24.058, Z 70.550}
   LaserStart_Ext()
   LIN {X -2.633, Y -23.682, Z 70.550} C_DIS
   LIN {X -3.182, Y -22.950, Z 70.550} C_DIS
   LIN {X -3.886, Y -22.018, Z 70.550} C_DIS
   LIN {X -4.123, Y -20.958, Z 70.550} C_DIS
   LIN {X -4.337, Y -19.981, Z 70.550} C_DIS
   LIN {X -4.110, Y -19.258, Z 70.550} C_DIS
   LIN {X -3.455, Y -17.088, Z 70.550} C_DIS
   LIN {X -2.769, Y -16.454, Z 70.550} C_DIS
   LIN {X -1.872, Y -15.598, Z 70.550} C_DIS
   LIN {X -0.204, Y -15.032, Z 70.550} C_DIS
   LIN {X 0.119, Y -14.926, Z 70.550} C_DIS
   LIN {X 0.371, Y -14.949, Z 70.550} C_DIS
   LIN {X 2.154, Y -15.102, Z 70.550} C_DIS
   LIN {X 3.845, Y -16.055, Z 70.550} C_DIS
   LIN {X 4.005, Y -16.145, Z 70.550} C_DIS
   LIN {X 4.130, Y -16.331, Z 70.550} C_DIS
   LIN {X 5.412, Y -18.263, Z 70.550} C_DIS
   LIN {X 5.628, Y -20.365, Z 70.550} C_DIS
   LIN {X 5.528, Y -20.752, Z 70.550} C_DIS
   LIN {X 4.788, Y -22.708, Z 70.550} C_DIS
   LIN {X 4.368, Y -23.114, Z 70.550} C_DIS
   LIN {X 3.297, Y -24.141, Z 70.550} C_DIS
   LIN {X 1.416, Y -24.797, Z 70.550} C_DIS
   LIN {X 1.210, Y -24.868, Z 70.550} C_DIS
   LIN {X 0.910, Y -24.841, Z 70.550} C_DIS
   LIN {X -0.829, Y -24.689, Z 70.550} C_DIS
   LIN {X -1.963, Y -24.058, Z 70.550}
   LaserEnd_Ext()
   LIN {X -4.415, Y -6.861, Z 70.550}
   LaserStart_Ext()
   LIN {X -4.307, Y -6.509, Z 70.550} C_DIS
   LIN {X -4.201, Y -6.058, Z 70.550} C_DIS
   LIN {X -3.291, Y -1.934, Z 70.550} C_DIS
   LIN {X -2.630, Y 2.538, Z 70.550} C_DIS
   LIN {X -2.349, Y 4.620, Z 70.550} C_DIS
   LIN {X -2.294, Y 6.038, Z 70.550} C_DIS
   LIN {X -2.210, Y 16.298, Z 70.550} C_DIS
   LIN {X -2.864, Y 22.454, Z 70.550} C_DIS
   LIN {X -3.154, Y 24.359, Z 70.550} C_DIS
   LIN {X -3.599, Y 26.484, Z 70.550} C_DIS
   LIN {X -3.959, Y 28.285, Z 70.550} C_DIS
   LIN {X -4.329, Y 29.700, Z 70.550} C_DIS
   LIN {X -5.021, Y 32.288, Z 70.550} C_DIS
   LIN {X -5.435, Y 33.587, Z 70.550} C_DIS
   LIN {X -5.901, Y 35.063, Z 70.550} C_DIS
   LIN {X -6.338, Y 36.288, Z 70.550} C_DIS
   LIN {X -6.700, Y 37.295, Z 70.550} C_DIS
   LIN {X -6.992, Y 38.046, Z 70.550} C_DIS
   LIN {X -7.279, Y 38.786, Z 70.550} C_DIS
   LIN {X -7.400, Y 39.089, Z 70.550} C_DIS
   LIN {X -7.747, Y 39.946, Z 70.550} C_DIS
   LIN {X -8.036, Y 41.363, Z 70.550} C_DIS
   LIN {X -8.069, Y 41.508, Z 70.550} C_DIS
   LIN {X -8.041, Y 41.708, Z 70.550} C_DIS
   LIN {X -7.900, Y 42.654, Z 70.550} C_DIS
   LIN {X -7.311, Y 43.707, Z 70.550} C_DIS
   LIN {X -7.073, Y 44.133, Z 70.550} C_DIS
   LIN {X -6.703, Y 44.483, Z 70.550} C_DIS
   LIN {X -4.947, Y 45.270, Z 70.550} C_DIS
   LIN {X -4.606, Y 45.443, Z 70.550} C_DIS
   LIN {X -4.184, Y 45.403, Z 70.550} C_DIS
   LIN {X -2.868, Y 45.281, Z 70.550} C_DIS
   LIN {X -2.000, Y 44.771, Z 70.550} C_DIS
   LIN {X -1.369, Y 44.398, Z 70.550} C_DIS
   LIN {X -0.868, Y 43.721, Z 70.550} C_DIS
   LIN {X -0.493, Y 43.216, Z 70.550} C_DIS
   LIN {X -0.281, Y 42.775, Z 70.550} C_DIS
   LIN {X 0.147, Y 41.877, Z 70.550} C_DIS
   LIN {X 0.917, Y 40.205, Z 70.550} C_DIS
   LIN {X 0.975, Y 40.078, Z 70.550} C_DIS
   LIN {X 1.555, Y 38.760, Z 70.550} C_DIS
   LIN {X 1.960, Y 37.817, Z 70.550} C_DIS
   LIN {X 2.689, Y 35.996, Z 70.550} C_DIS
   LIN {X 3.341, Y 34.396, Z 70.550} C_DIS
   LIN {X 3.866, Y 32.978, Z 70.550} C_DIS
   LIN {X 4.519, Y 31.194, Z 70.550} C_DIS
   LIN {X 5.367, Y 28.587, Z 70.550} C_DIS
   LIN {X 6.171, Y 26.073, Z 70.550} C_DIS
   LIN {X 7.788, Y 19.932, Z 70.550} C_DIS
   LIN {X 9.195, Y 12.641, Z 70.550} C_DIS
   LIN {X 9.878, Y 8.254, Z 70.550} C_DIS
   LIN {X 10.360, Y 3.983, Z 70.550} C_DIS
   LIN {X 10.428, Y 2.887, Z 70.550} C_DIS
   LIN {X 10.596, Y 0.151, Z 70.550} C_DIS
   LIN {X 10.726, Y -6.364, Z 70.550} C_DIS
   LIN {X 10.645, Y -9.202, Z 70.550} C_DIS
   LIN {X 10.576, Y -11.150, Z 70.550} C_DIS
   LIN {X 10.314, Y -14.888, Z 70.550} C_DIS
   LIN {X 10.301, Y -15.031, Z 70.550} C_DIS
   LIN {X 10.011, Y -17.892, Z 70.550} C_DIS
   LIN {X 9.776, Y -19.752, Z 70.550} C_DIS
   LIN {X 9.594, Y -21.129, Z 70.550} C_DIS
   LIN {X 8.983, Y -23.033, Z 70.550} C_DIS
   LIN {X 8.692, Y -23.950, Z 70.550} C_DIS
   LIN {X 8.295, Y -24.493, Z 70.550} C_DIS
   LIN {X 6.788, Y -26.470, Z 70.550} C_DIS
   LIN {X 3.833, Y -28.199, Z 70.550} C_DIS
   LIN {X 3.301, Y -28.502, Z 70.550} C_DIS
   LIN {X 2.105, Y -28.647, Z 70.550} C_DIS
   LIN {X 0.112, Y -28.897, Z 70.550} C_DIS
   LIN {X -0.714, Y -28.687, Z 70.550} C_DIS
   LIN {X -3.433, Y -27.954, Z 70.550} C_DIS
   LIN {X -4.985, Y -26.842, Z 70.550} C_DIS
   LIN {X -5.672, Y -26.354, Z 70.550} C_DIS
   LIN {X -6.324, Y -25.357, Z 70.550} C_DIS
   LIN {X -7.736, Y -23.223, Z 70.550} C_DIS
   LIN {X -8.303, Y -19.792, Z 70.550} C_DIS
   LIN {X -8.340, Y -19.563, Z 70.550} C_DIS
   LIN {X -8.300, Y -19.389, Z 70.550} C_DIS
   LIN {X -7.648, Y -16.468, Z 70.550} C_DIS
   LIN {X -6.628, Y -13.885, Z 70.550} C_DIS
   LIN {X -6.538, Y -13.651, Z 70.550} C_DIS
   LIN {X -5.638, Y -11.066, Z 70.550} C_DIS
   LIN {X -4.415, Y -6.861, Z 70.550}
   LaserEnd_Ext()
   LIN {X -7.280, Y -19.851, Z 70.550}
   LaserStart_Ext()
   LIN {X -7.280, Y -19.408, Z 70.550}
   LaserEnd_Ext()
   LIN {X -6.280, Y 43.502, Z 70.550}
   LaserStart_Ext()
   LIN {X -6.280, Y 38.976, Z 70.550}
   LaserEnd_Ext()
   LIN {X -6.280, Y -15.727, Z 70.550}
   LaserStart_Ext()
   LIN {X -6.280, Y -23.612, Z 70.550}
   LaserEnd_Ext()
   LIN {X -5.280, Y -25.127, Z 70.550}
   LaserStart_Ext()
   LIN {X -5.280, Y -20.352, Z 70.550}
   LaserEnd_Ext()
   LIN {X -5.280, Y -19.644, Z 70.550}
   LaserStart_Ext()
   LIN {X -5.280, Y -13.078, Z 70.550}
   LaserEnd_Ext()
   LIN {X -5.280, Y 36.297, Z 70.550}
   LaserStart_Ext()
   LIN {X -5.280, Y 44.025, Z 70.550}
   LaserEnd_Ext()
   LIN {X -4.280, Y 44.408, Z 70.550}
   LaserStart_Ext()
   LIN {X -4.280, Y 33.256, Z 70.550}
   LaserEnd_Ext()
   LIN {X -4.280, Y -9.975, Z 70.550}
   LaserStart_Ext()
   LIN {X -4.280, Y -16.524, Z 70.550}
   LaserEnd_Ext()
   LIN {X -4.280, Y -23.156, Z 70.550}
   LaserStart_Ext()
   LIN {X -4.280, Y -26.117, Z 70.550}
   LaserEnd_Ext()
   LIN {X -3.280, Y -26.833, Z 70.550}
   LaserStart_Ext()
   LIN {X -3.280, Y -24.444, Z 70.550}
   LaserEnd_Ext()
   LIN {X -3.280, Y -15.559, Z 70.550}
   LaserStart_Ext()
   LIN {X -3.280, Y -6.509, Z 70.550}
   LaserEnd_Ext()
   LIN {X -3.280, Y 29.640, Z 70.550}
   LaserStart_Ext()
   LIN {X -3.280, Y 44.315, Z 70.550}
   LaserEnd_Ext()
   LIN {X -2.280, Y 43.775, Z 70.550}
   LaserStart_Ext()
   LIN {X -2.280, Y 25.066, Z 70.550}
   LaserEnd_Ext()
   LIN {X -2.280, Y -1.933, Z 70.550}
   LaserStart_Ext()
   LIN {X -2.280, Y -14.686, Z 70.550}
   LaserEnd_Ext()
   LIN {X -2.280, Y -25.026, Z 70.550}
   LaserStart_Ext()
   LIN {X -2.280, Y -27.229, Z 70.550}
   LaserEnd_Ext()
   LIN {X -1.280, Y -27.499, Z 70.550}
   LaserStart_Ext()
   LIN {X -1.280, Y -25.580, Z 70.550}
   LaserEnd_Ext()
   LIN {X -1.280, Y -14.341, Z 70.550}
   LaserStart_Ext()
   LIN {X -1.280, Y 7.788, Z 70.550}
   LaserEnd_Ext()
   LIN {X -1.280, Y 17.007, Z 70.550}
   LaserStart_Ext()
   LIN {X -1.280, Y 42.545, Z 70.550}
   LaserEnd_Ext()
   LIN {X -0.280, Y 40.414, Z 70.550}
   LaserStart_Ext()
   LIN {X -0.280, Y -14.005, Z 70.550}
   LaserEnd_Ext()
   LIN {X -0.280, Y -25.740, Z 70.550}
   LaserStart_Ext()
   LIN {X -0.280, Y -27.766, Z 70.550}
   LaserEnd_Ext()
   LIN {X 0.720, Y -27.813, Z 70.550}
   LaserStart_Ext()
   LIN {X 0.720, Y -25.828, Z 70.550}
   LaserEnd_Ext()
   LIN {X 0.720, Y -13.975, Z 70.550}
   LaserStart_Ext()
   LIN {X 0.720, Y 38.170, Z 70.550}
   LaserEnd_Ext()
   LIN {X 1.720, Y 35.726, Z 70.550}
   LaserStart_Ext()
   LIN {X 1.720, Y -14.061, Z 70.550}
   LaserEnd_Ext()
   LIN {X 1.720, Y -25.750, Z 70.550}
   LaserStart_Ext()
   LIN {X 1.720, Y -27.687, Z 70.550}
   LaserEnd_Ext()
   LIN {X 2.720, Y -27.565, Z 70.550}
   LaserStart_Ext()
   LIN {X 2.720, Y -25.401, Z 70.550}
   LaserEnd_Ext()
   LIN {X 2.720, Y -14.274, Z 70.550}
   LaserStart_Ext()
   LIN {X 2.720, Y 33.194, Z 70.550}
   LaserEnd_Ext()
   LIN {X 3.720, Y 30.417, Z 70.550}
   LaserStart_Ext()
   LIN {X 3.720, Y -14.837, Z 70.550}
   LaserEnd_Ext()
   LIN {X 3.720, Y -25.047, Z 70.550}
   LaserStart_Ext()
   LIN {X 3.720, Y -27.107, Z 70.550}
   LaserEnd_Ext()
   LIN {X 4.720, Y -26.521, Z 70.550}
   LaserStart_Ext()
   LIN {X 4.720, Y -24.162, Z 70.550}
   LaserEnd_Ext()
   LIN {X 4.720, Y -15.445, Z 70.550}
   LaserStart_Ext()
   LIN {X 4.720, Y 27.327, Z 70.550}
   LaserEnd_Ext()
   LIN {X 5.720, Y 23.858, Z 70.550}
   LaserStart_Ext()
   LIN {X 5.720, Y -16.918, Z 70.550}
   LaserEnd_Ext()
   LIN {X 5.720, Y -23.069, Z 70.550}
   LaserStart_Ext()
   LIN {X 5.720, Y -25.936, Z 70.550}
   LaserEnd_Ext()
   LIN {X 6.720, Y -24.910, Z 70.550}
   LaserStart_Ext()
   LIN {X 6.720, Y 20.060, Z 70.550}
   LaserEnd_Ext()
   LIN {X 7.720, Y 15.006, Z 70.550}
   LaserStart_Ext()
   LIN {X 7.720, Y -23.586, Z 70.550}
   LaserEnd_Ext()
   LIN {X 8.720, Y -20.110, Z 70.550}
   LaserStart_Ext()
   LIN {X 8.720, Y 9.190, Z 70.550}
   LaserEnd_Ext()
   LIN {X 9.720, Y -6.089, Z 70.550}
   LaserStart_Ext()
   LIN {X 9.720, Y -6.549, Z 70.550}
   LaserEnd_Ext()
   LIN {X 1.304, Y -24.812, Z 71.400}
   LaserStart_Ext()
   LIN {X 0.229, Y -24.723, Z 71.400} C_DIS
   LIN {X -0.738, Y -24.638, Z 71.400} C_DIS
   LIN {X -1.883, Y -24.002, Z 71.400} C_DIS
   LIN {X -2.545, Y -23.636, Z 71.400} C_DIS
   LIN {X -2.899, Y -23.172, Z 71.400} C_DIS
   LIN {X -3.802, Y -21.975, Z 71.400} C_DIS
   LIN {X -4.151, Y -20.409, Z 71.400} C_DIS
   LIN {X -4.258, Y -19.939, Z 71.400} C_DIS
   LIN {X -3.479, Y -17.357, Z 71.400} C_DIS
   LIN {X -3.394, Y -17.061, Z 71.400} C_DIS
   LIN {X -2.997, Y -16.674, Z 71.400} C_DIS
   LIN {X -1.851, Y -15.579, Z 71.400} C_DIS
   LIN {X -0.868, Y -15.246, Z 71.400} C_DIS
   LIN {X 0.152, Y -14.879, Z 71.400} C_DIS
   LIN {X 1.497, Y -14.983, Z 71.400} C_DIS
   LIN {X 2.222, Y -15.045, Z 71.400} C_DIS
   LIN {X 2.741, Y -15.338, Z 71.400} C_DIS
   LIN {X 4.076, Y -16.083, Z 71.400} C_DIS
   LIN {X 5.110, Y -17.629, Z 71.400} C_DIS
   LIN {X 5.488, Y -18.198, Z 71.400} C_DIS
   LIN {X 5.558, Y -18.880, Z 71.400} C_DIS
   LIN {X 5.719, Y -20.396, Z 71.400} C_DIS
   LIN {X 5.368, Y -21.337, Z 71.400} C_DIS
   LIN {X 4.874, Y -22.645, Z 71.400} C_DIS
   LIN {X 3.576, Y -23.900, Z 71.400} C_DIS
   LIN {X 3.389, Y -24.079, Z 71.400} C_DIS
   LIN {X 2.968, Y -24.226, Z 71.400} C_DIS
   LIN {X 1.304, Y -24.812, Z 71.400}
   LaserEnd_Ext()
   LIN {X 0.082, Y 41.929, Z 71.400}
   LaserStart_Ext()
   LIN {X 0.233, Y 41.606, Z 71.400} C_DIS
   LIN {X 0.888, Y 40.190, Z 71.400} C_DIS
   LIN {X 1.807, Y 38.102, Z 71.400} C_DIS
   LIN {X 1.867, Y 37.962, Z 71.400} C_DIS
   LIN {X 1.975, Y 37.692, Z 71.400} C_DIS
   LIN {X 3.258, Y 34.546, Z 71.400} C_DIS
   LIN {X 4.291, Y 31.756, Z 71.400} C_DIS
   LIN {X 4.581, Y 30.963, Z 71.400} C_DIS
   LIN {X 4.958, Y 29.804, Z 71.400} C_DIS
   LIN {X 6.297, Y 25.616, Z 71.400} C_DIS
   LIN {X 7.750, Y 20.097, Z 71.400} C_DIS
   LIN {X 9.399, Y 11.553, Z 71.400} C_DIS
   LIN {X 9.867, Y 8.548, Z 71.400} C_DIS
   LIN {X 10.415, Y 3.699, Z 71.400} C_DIS
   LIN {X 10.491, Y 2.454, Z 71.400} C_DIS
   LIN {X 10.628, Y 0.228, Z 71.400} C_DIS
   LIN {X 10.686, Y -1.909, Z 71.400} C_DIS
   LIN {X 10.773, Y -6.286, Z 71.400} C_DIS
   LIN {X 10.646, Y -10.768, Z 71.400} C_DIS
   LIN {X 10.635, Y -11.072, Z 71.400} C_DIS
   LIN {X 10.592, Y -11.689, Z 71.400} C_DIS
   LIN {X 10.377, Y -14.869, Z 71.400} C_DIS
   LIN {X 10.264, Y -16.060, Z 71.400} C_DIS
   LIN {X 10.086, Y -17.816, Z 71.400} C_DIS
   LIN {X 9.699, Y -20.879, Z 71.400} C_DIS
   LIN {X 9.676, Y -21.054, Z 71.400} C_DIS
   LIN {X 9.598, Y -21.296, Z 71.400} C_DIS
   LIN {X 8.781, Y -23.877, Z 71.400} C_DIS
   LIN {X 7.664, Y -25.406, Z 71.400} C_DIS
   LIN {X 6.958, Y -26.331, Z 71.400} C_DIS
   LIN {X 4.813, Y -27.587, Z 71.400} C_DIS
   LIN {X 3.431, Y -28.430, Z 71.400} C_DIS
   LIN {X 2.813, Y -28.534, Z 71.400} C_DIS
   LIN {X 0.315, Y -28.848, Z 71.400} C_DIS
   LIN {X -1.606, Y -28.359, Z 71.400} C_DIS
   LIN {X -3.406, Y -27.874, Z 71.400} C_DIS
   LIN {X -5.392, Y -26.450, Z 71.400} C_DIS
   LIN {X -5.602, Y -26.291, Z 71.400} C_DIS
   LIN {X -5.735, Y -26.082, Z 71.400} C_DIS
   LIN {X -7.649, Y -23.189, Z 71.400} C_DIS
   LIN {X -8.093, Y -20.507, Z 71.400} C_DIS
   LIN {X -8.262, Y -19.530, Z 71.400} C_DIS
   LIN {X -7.958, Y -18.138, Z 71.400} C_DIS
   LIN {X -7.577, Y -16.434, Z 71.400} C_DIS
   LIN {X -7.046, Y -15.090, Z 71.400} C_DIS
   LIN {X -6.404, Y -13.416, Z 71.400} C_DIS
   LIN {X -5.711, Y -11.426, Z 71.400} C_DIS
   LIN {X -4.770, Y -8.189, Z 71.400} C_DIS
   LIN {X -4.365, Y -6.873, Z 71.400} C_DIS
   LIN {X -3.968, Y -5.186, Z 71.400} C_DIS
   LIN {X -3.334, Y -2.313, Z 71.400} C_DIS
   LIN {X -2.511, Y 3.252, Z 71.400} C_DIS
   LIN {X -2.349, Y 4.458, Z 71.400} C_DIS
   LIN {X -2.317, Y 5.280, Z 71.400} C_DIS
   LIN {X -2.225, Y 16.514, Z 71.400} C_DIS
   LIN {X -2.782, Y 21.761, Z 71.400} C_DIS
   LIN {X -3.214, Y 24.600, Z 71.400} C_DIS
   LIN {X -3.877, Y 27.767, Z 71.400} C_DIS
   LIN {X -3.968, Y 28.220, Z 71.400} C_DIS
   LIN {X -4.061, Y 28.576, Z 71.400} C_DIS
   LIN {X -4.169, Y 28.978, Z 71.400} C_DIS
   LIN {X -5.064, Y 32.328, Z 71.400} C_DIS
   LIN {X -5.438, Y 33.501, Z 71.400} C_DIS
   LIN {X -5.951, Y 35.101, Z 71.400} C_DIS
   LIN {X -6.402, Y 36.348, Z 71.400} C_DIS
   LIN {X -6.754, Y 37.331, Z 71.400} C_DIS
   LIN {X -6.988, Y 37.930, Z 71.400} C_DIS
   LIN {X -7.337, Y 38.821, Z 71.400} C_DIS
   LIN {X -7.730, Y 39.786, Z 71.400} C_DIS
   LIN {X -7.808, Y 39.980, Z 71.400} C_DIS
   LIN {X -7.840, Y 40.135, Z 71.400} C_DIS
   LIN {X -8.128, Y 41.390, Z 71.400} C_DIS
   LIN {X -7.985, Y 42.423, Z 71.400} C_DIS
   LIN {X -7.957, Y 42.720, Z 71.400} C_DIS
   LIN {X -7.812, Y 43.008, Z 71.400} C_DIS
   LIN {X -7.198, Y 44.104, Z 71.400} C_DIS
   LIN {X -6.631, Y 44.645, Z 71.400} C_DIS
   LIN {X -6.553, Y 44.719, Z 71.400} C_DIS
   LIN {X -6.269, Y 44.846, Z 71.400} C_DIS
   LIN {X -4.679, Y 45.484, Z 71.400} C_DIS
   LIN {X -3.616, Y 45.389, Z 71.400} C_DIS
   LIN {X -2.941, Y 45.326, Z 71.400} C_DIS
   LIN {X -2.192, Y 44.886, Z 71.400} C_DIS
   LIN {X -1.440, Y 44.447, Z 71.400} C_DIS
   LIN {X -1.043, Y 43.915, Z 71.400} C_DIS
   LIN {X -0.561, Y 43.267, Z 71.400} C_DIS
   LIN {X -0.098, Y 42.302, Z 71.400} C_DIS
   LIN {X 0.082, Y 41.929, Z 71.400}
   LaserEnd_Ext()
   LIN {X -1.469, Y -27.360, Z 71.400}
   LaserStart_Ext()
   LIN {X 3.265, Y -27.360, Z 71.400}
   LaserEnd_Ext()
   LIN {X 4.930, Y -26.360, Z 71.400}
   LaserStart_Ext()
   LIN {X -3.801, Y -26.360, Z 71.400}
   LaserEnd_Ext()
   LIN {X -5.013, Y -25.360, Z 71.400}
   LaserStart_Ext()
   LIN {X -1.498, Y -25.360, Z 71.400}
   LaserEnd_Ext()
   LIN {X 2.759, Y -25.360, Z 71.400}
   LaserStart_Ext()
   LIN {X 6.441, Y -25.360, Z 71.400}
   LaserEnd_Ext()
   LIN {X 7.190, Y -24.360, Z 71.400}
   LaserStart_Ext()
   LIN {X 4.539, Y -24.360, Z 71.400}
   LaserEnd_Ext()
   LIN {X -3.233, Y -24.360, Z 71.400}
   LaserStart_Ext()
   LIN {X -5.675, Y -24.360, Z 71.400}
   LaserEnd_Ext()
   LIN {X -6.337, Y -23.360, Z 71.400}
   LaserStart_Ext()
   LIN {X -4.009, Y -23.360, Z 71.400}
   LaserEnd_Ext()
   LIN {X 5.572, Y -23.360, Z 71.400}
   LaserStart_Ext()
   LIN {X 7.896, Y -23.360, Z 71.400}
   LaserEnd_Ext()
   LIN {X 8.212, Y -22.360, Z 71.400}
   LaserStart_Ext()
   LIN {X 6.050, Y -22.360, Z 71.400}
   LaserEnd_Ext()
   LIN {X -4.723, Y -22.360, Z 71.400}
   LaserStart_Ext()
   LIN {X -6.773, Y -22.360, Z 71.400}
   LaserEnd_Ext()
   LIN {X -6.938, Y -21.360, Z 71.400}
   LaserStart_Ext()
   LIN {X -4.964, Y -21.360, Z 71.400}
   LaserEnd_Ext()
   LIN {X 6.427, Y -21.360, Z 71.400}
   LaserStart_Ext()
   LIN {X 8.529, Y -21.360, Z 71.400}
   LaserEnd_Ext()
   LIN {X 8.757, Y -20.360, Z 71.400}
   LaserStart_Ext()
   LIN {X 6.717, Y -20.360, Z 71.400}
   LaserEnd_Ext()
   LIN {X -5.188, Y -20.360, Z 71.400}
   LaserStart_Ext()
   LIN {X -7.103, Y -20.360, Z 71.400}
   LaserEnd_Ext()
   LIN {X -7.201, Y -19.360, Z 71.400}
   LaserStart_Ext()
   LIN {X -5.128, Y -19.360, Z 71.400}
   LaserEnd_Ext()
   LIN {X 6.614, Y -19.360, Z 71.400}
   LaserStart_Ext()
   LIN {X 8.883, Y -19.360, Z 71.400}
   LaserEnd_Ext()
   LIN {X 9.009, Y -18.360, Z 71.400}
   LaserStart_Ext()
   LIN {X 6.510, Y -18.360, Z 71.400}
   LaserEnd_Ext()
   LIN {X -4.827, Y -18.360, Z 71.400}
   LaserStart_Ext()
   LIN {X -6.982, Y -18.360, Z 71.400}
   LaserEnd_Ext()
   LIN {X -6.759, Y -17.360, Z 71.400}
   LaserStart_Ext()
   LIN {X -4.525, Y -17.360, Z 71.400}
   LaserEnd_Ext()
   LIN {X 6.132, Y -17.360, Z 71.400}
   LaserStart_Ext()
   LIN {X 9.127, Y -17.360, Z 71.400}
   LaserEnd_Ext()
   LIN {X 9.228, Y -16.360, Z 71.400}
   LaserStart_Ext()
   LIN {X 5.465, Y -16.360, Z 71.400}
   LaserEnd_Ext()
   LIN {X -4.106, Y -16.360, Z 71.400}
   LaserStart_Ext()
   LIN {X -6.472, Y -16.360, Z 71.400}
   LaserEnd_Ext()
   LIN {X -6.079, Y -15.360, Z 71.400}
   LaserStart_Ext()
   LIN {X -3.069, Y -15.360, Z 71.400}
   LaserEnd_Ext()
   LIN {X 4.766, Y -15.360, Z 71.400}
   LaserStart_Ext()
   LIN {X 9.326, Y -15.360, Z 71.400}
   LaserEnd_Ext()
   LIN {X 9.409, Y -14.360, Z 71.400}
   LaserStart_Ext()
   LIN {X 3.043, Y -14.360, Z 71.400}
   LaserEnd_Ext()
   LIN {X -1.370, Y -14.360, Z 71.400}
   LaserStart_Ext()
   LIN {X -5.695, Y -14.360, Z 71.400}
   LaserEnd_Ext()
   LIN {X -5.326, Y -13.360, Z 71.400}
   LaserStart_Ext()
   LIN {X 9.477, Y -13.360, Z 71.400}
   LaserEnd_Ext()
   LIN {X 9.544, Y -12.360, Z 71.400}
   LaserStart_Ext()
   LIN {X -4.978, Y -12.360, Z 71.400}
   LaserEnd_Ext()
   LIN {X -4.651, Y -11.360, Z 71.400}
   LaserStart_Ext()
   LIN {X 9.612, Y -11.360, Z 71.400}
   LaserEnd_Ext()
   LIN {X 9.657, Y -10.360, Z 71.400}
   LaserStart_Ext()
   LIN {X -4.360, Y -10.360, Z 71.400}
   LaserEnd_Ext()
   LIN {X -4.069, Y -9.360, Z 71.400}
   LaserStart_Ext()
   LIN {X 9.685, Y -9.360, Z 71.400}
   LaserEnd_Ext()
   LIN {X 9.714, Y -8.360, Z 71.400}
   LaserStart_Ext()
   LIN {X -3.776, Y -8.360, Z 71.400}
   LaserEnd_Ext()
   LIN {X -3.469, Y -7.360, Z 71.400}
   LaserStart_Ext()
   LIN {X 9.742, Y -7.360, Z 71.400}
   LaserEnd_Ext()
   LIN {X 9.771, Y -6.360, Z 71.400}
   LaserStart_Ext()
   LIN {X -3.217, Y -6.360, Z 71.400}
   LaserEnd_Ext()
   LIN {X -2.982, Y -5.360, Z 71.400}
   LaserStart_Ext()
   LIN {X 9.755, Y -5.360, Z 71.400}
   LaserEnd_Ext()
   LIN {X 9.735, Y -4.360, Z 71.400}
   LaserStart_Ext()
   LIN {X -2.762, Y -4.360, Z 71.400}
   LaserEnd_Ext()
   LIN {X -2.541, Y -3.360, Z 71.400}
   LaserStart_Ext()
   LIN {X 9.715, Y -3.360, Z 71.400}
   LaserEnd_Ext()
   LIN {X 9.695, Y -2.360, Z 71.400}
   LaserStart_Ext()
   LIN {X -2.330, Y -2.360, Z 71.400}
   LaserEnd_Ext()
   LIN {X -2.182, Y -1.360, Z 71.400}
   LaserStart_Ext()
   LIN {X 9.671, Y -1.360, Z 71.400}
   LaserEnd_Ext()
   LIN {X 9.644, Y -0.360, Z 71.400}
   LaserStart_Ext()
   LIN {X -2.035, Y -0.360, Z 71.400}
   LaserEnd_Ext()
   LIN {X -1.887, Y 0.640, Z 71.400}
   LaserStart_Ext()
   LIN {X 9.601, Y 0.640, Z 71.400}
   LaserEnd_Ext()
   LIN {X 9.539, Y 1.640, Z 71.400}
   LaserStart_Ext()
   LIN {X -1.739, Y 1.640, Z 71.400}
   LaserEnd_Ext()
   LIN {X -1.591, Y 2.640, Z 71.400}
   LaserStart_Ext()
   LIN {X 9.478, Y 2.640, Z 71.400}
   LaserEnd_Ext()
   LIN {X 9.415, Y 3.640, Z 71.400}
   LaserStart_Ext()
   LIN {X -1.450, Y 3.640, Z 71.400}
   LaserEnd_Ext()
   LIN {X -1.341, Y 4.640, Z 71.400}
   LaserStart_Ext()
   LIN {X 9.302, Y 4.640, Z 71.400}
   LaserEnd_Ext()
   LIN {X 9.189, Y 5.640, Z 71.400}
   LaserStart_Ext()
   LIN {X -1.314, Y 5.640, Z 71.400}
   LaserEnd_Ext()
   LIN {X -1.306, Y 6.640, Z 71.400}
   LaserStart_Ext()
   LIN {X 9.076, Y 6.640, Z 71.400}
   LaserEnd_Ext()
   LIN {X 8.963, Y 7.640, Z 71.400}
   LaserStart_Ext()
   LIN {X -1.298, Y 7.640, Z 71.400}
   LaserEnd_Ext()
   LIN {X -1.289, Y 8.640, Z 71.400}
   LaserStart_Ext()
   LIN {X 8.841, Y 8.640, Z 71.400}
   LaserEnd_Ext()
   LIN {X 8.685, Y 9.640, Z 71.400}
   LaserStart_Ext()
   LIN {X -1.281, Y 9.640, Z 71.400}
   LaserEnd_Ext()
   LIN {X -1.273, Y 10.640, Z 71.400}
   LaserStart_Ext()
   LIN {X 8.529, Y 10.640, Z 71.400}
   LaserEnd_Ext()
   LIN {X 8.364, Y 11.640, Z 71.400}
   LaserStart_Ext()
   LIN {X -1.265, Y 11.640, Z 71.400}
   LaserEnd_Ext()
   LIN {X -1.257, Y 12.640, Z 71.400}
   LaserStart_Ext()
   LIN {X 8.171, Y 12.640, Z 71.400}
   LaserEnd_Ext()
   LIN {X 7.978, Y 13.640, Z 71.400}
   LaserStart_Ext()
   LIN {X -1.248, Y 13.640, Z 71.400}
   LaserEnd_Ext()
   LIN {X -1.240, Y 14.640, Z 71.400}
   LaserStart_Ext()
   LIN {X 7.785, Y 14.640, Z 71.400}
   LaserEnd_Ext()
   LIN {X 7.592, Y 15.640, Z 71.400}
   LaserStart_Ext()
   LIN {X -1.232, Y 15.640, Z 71.400}
   LaserEnd_Ext()
   LIN {X -1.233, Y 16.640, Z 71.400}
   LaserStart_Ext()
   LIN {X 7.399, Y 16.640, Z 71.400}
   LaserEnd_Ext()
   LIN {X 7.206, Y 17.640, Z 71.400}
   LaserStart_Ext()
   LIN {X -1.339, Y 17.640, Z 71.400}
   LaserEnd_Ext()
   LIN {X -1.445, Y 18.640, Z 71.400}
   LaserStart_Ext()
   LIN {X 7.013, Y 18.640, Z 71.400}
   LaserEnd_Ext()
   LIN {X 6.820, Y 19.640, Z 71.400}
   LaserStart_Ext()
   LIN {X -1.551, Y 19.640, Z 71.400}
   LaserEnd_Ext()
   LIN {X -1.658, Y 20.640, Z 71.400}
   LaserStart_Ext()
   LIN {X 6.573, Y 20.640, Z 71.400}
   LaserEnd_Ext()
   LIN {X 6.310, Y 21.640, Z 71.400}
   LaserStart_Ext()
   LIN {X -1.764, Y 21.640, Z 71.400}
   LaserEnd_Ext()
   LIN {X -1.904, Y 22.640, Z 71.400}
   LaserStart_Ext()
   LIN {X 6.047, Y 22.640, Z 71.400}
   LaserEnd_Ext()
   LIN {X 5.783, Y 23.640, Z 71.400}
   LaserStart_Ext()
   LIN {X -2.056, Y 23.640, Z 71.400}
   LaserEnd_Ext()
   LIN {X -2.208, Y 24.640, Z 71.400}
   LaserStart_Ext()
   LIN {X 5.520, Y 24.640, Z 71.400}
   LaserEnd_Ext()
   LIN {X 5.240, Y 25.640, Z 71.400}
   LaserStart_Ext()
   LIN {X -2.410, Y 25.640, Z 71.400}
   LaserEnd_Ext()
   LIN {X -2.619, Y 26.640, Z 71.400}
   LaserStart_Ext()
   LIN {X 4.920, Y 26.640, Z 71.400}
   LaserEnd_Ext()
   LIN {X 4.600, Y 27.640, Z 71.400}
   LaserStart_Ext()
   LIN {X -2.829, Y 27.640, Z 71.400}
   LaserEnd_Ext()
   LIN {X -3.044, Y 28.640, Z 71.400}
   LaserStart_Ext()
   LIN {X 4.280, Y 28.640, Z 71.400}
   LaserEnd_Ext()
   LIN {X 3.960, Y 29.640, Z 71.400}
   LaserStart_Ext()
   LIN {X -3.310, Y 29.640, Z 71.400}
   LaserEnd_Ext()
   LIN {X -3.578, Y 30.640, Z 71.400}
   LaserStart_Ext()
   LIN {X 3.634, Y 30.640, Z 71.400}
   LaserEnd_Ext()
   LIN {X 3.268, Y 31.640, Z 71.400}
   LaserStart_Ext()
   LIN {X -3.845, Y 31.640, Z 71.400}
   LaserEnd_Ext()
   LIN {X -4.114, Y 32.640, Z 71.400}
   LaserStart_Ext()
   LIN {X 2.897, Y 32.640, Z 71.400}
   LaserEnd_Ext()
   LIN {X 2.527, Y 33.640, Z 71.400}
   LaserStart_Ext()
   LIN {X -4.432, Y 33.640, Z 71.400}
   LaserEnd_Ext()
   LIN {X -4.753, Y 34.640, Z 71.400}
   LaserStart_Ext()
   LIN {X 2.140, Y 34.640, Z 71.400}
   LaserEnd_Ext()
   LIN {X 1.732, Y 35.640, Z 71.400}
   LaserStart_Ext()
   LIN {X -5.082, Y 35.640, Z 71.400}
   LaserEnd_Ext()
   LIN {X -5.444, Y 36.640, Z 71.400}
   LaserStart_Ext()
   LIN {X 1.324, Y 36.640, Z 71.400}
   LaserEnd_Ext()
   LIN {X 0.917, Y 37.640, Z 71.400}
   LaserStart_Ext()
   LIN {X -5.803, Y 37.640, Z 71.400}
   LaserEnd_Ext()
   LIN {X -6.192, Y 38.640, Z 71.400}
   LaserStart_Ext()
   LIN {X 0.478, Y 38.640, Z 71.400}
   LaserEnd_Ext()
   LIN {X 0.037, Y 39.640, Z 71.400}
   LaserStart_Ext()
   LIN {X -6.591, Y 39.640, Z 71.400}
   LaserEnd_Ext()
   LIN {X -6.930, Y 40.640, Z 71.400}
   LaserStart_Ext()
   LIN {X -0.422, Y 40.640, Z 71.400}
   LaserEnd_Ext()
   LIN {X -0.889, Y 41.640, Z 71.400}
   LaserStart_Ext()
   LIN {X -7.084, Y 41.640, Z 71.400}
   LaserEnd_Ext()
   LIN {X -6.872, Y 42.640, Z 71.400}
   LaserStart_Ext()
   LIN {X -1.370, Y 42.640, Z 71.400}
   LaserEnd_Ext()
   LIN {X -2.085, Y 43.640, Z 71.400}
   LaserStart_Ext()
   LIN {X -6.236, Y 43.640, Z 71.400}
   LaserEnd_Ext()
   LIN {X 2.529, Y -24.358, Z 72.250}
   LaserStart_Ext()
   LIN {X 1.398, Y -24.757, Z 72.250} C_DIS
   LIN {X -0.221, Y -24.622, Z 72.250} C_DIS
   LIN {X -0.648, Y -24.588, Z 72.250} C_DIS
   LIN {X -0.918, Y -24.440, Z 72.250} C_DIS
   LIN {X -2.457, Y -23.590, Z 72.250} C_DIS
   LIN {X -3.622, Y -22.058, Z 72.250} C_DIS
   LIN {X -3.717, Y -21.932, Z 72.250} C_DIS
   LIN {X -3.754, Y -21.767, Z 72.250} C_DIS
   LIN {X -4.179, Y -19.897, Z 72.250} C_DIS
   LIN {X -3.728, Y -18.402, Z 72.250} C_DIS
   LIN {X -3.333, Y -17.034, Z 72.250} C_DIS
   LIN {X -2.020, Y -15.753, Z 72.250} C_DIS
   LIN {X -1.825, Y -15.558, Z 72.250} C_DIS
   LIN {X -1.492, Y -15.433, Z 72.250} C_DIS
   LIN {X 0.177, Y -14.832, Z 72.250} C_DIS
   LIN {X 1.569, Y -14.940, Z 72.250} C_DIS
   LIN {X 2.290, Y -14.987, Z 72.250} C_DIS
   LIN {X 3.037, Y -15.402, Z 72.250} C_DIS
   LIN {X 4.146, Y -16.021, Z 72.250} C_DIS
   LIN {X 4.976, Y -17.261, Z 72.250} C_DIS
   LIN {X 5.563, Y -18.133, Z 72.250} C_DIS
   LIN {X 5.650, Y -18.925, Z 72.250} C_DIS
   LIN {X 5.799, Y -20.330, Z 72.250} C_DIS
   LIN {X 5.071, Y -22.285, Z 72.250} C_DIS
   LIN {X 4.959, Y -22.582, Z 72.250} C_DIS
   LIN {X 4.557, Y -22.971, Z 72.250} C_DIS
   LIN {X 3.479, Y -24.019, Z 72.250} C_DIS
   LIN {X 2.529, Y -24.358, Z 72.250}
   LaserEnd_Ext()
   LIN {X -4.993, Y 45.429, Z 72.250}
   LaserStart_Ext()
   LIN {X -4.753, Y 45.525, Z 72.250} C_DIS
   LIN {X -4.396, Y 45.493, Z 72.250} C_DIS
   LIN {X -3.015, Y 45.371, Z 72.250} C_DIS
   LIN {X -2.378, Y 45.002, Z 72.250} C_DIS
   LIN {X -1.511, Y 44.495, Z 72.250} C_DIS
   LIN {X -0.953, Y 43.747, Z 72.250} C_DIS
   LIN {X -0.630, Y 43.317, Z 72.250} C_DIS
   LIN {X -0.423, Y 42.891, Z 72.250} C_DIS
   LIN {X 0.016, Y 41.981, Z 72.250} C_DIS
   LIN {X 0.814, Y 40.270, Z 72.250} C_DIS
   LIN {X 1.523, Y 38.663, Z 72.250} C_DIS
   LIN {X 1.868, Y 37.889, Z 72.250} C_DIS
   LIN {X 2.506, Y 36.335, Z 72.250} C_DIS
   LIN {X 3.175, Y 34.695, Z 72.250} C_DIS
   LIN {X 4.316, Y 31.612, Z 72.250} C_DIS
   LIN {X 4.561, Y 30.953, Z 72.250} C_DIS
   LIN {X 4.630, Y 30.772, Z 72.250} C_DIS
   LIN {X 4.699, Y 30.551, Z 72.250} C_DIS
   LIN {X 6.423, Y 25.160, Z 72.250} C_DIS
   LIN {X 7.712, Y 20.263, Z 72.250} C_DIS
   LIN {X 9.604, Y 10.464, Z 72.250} C_DIS
   LIN {X 9.856, Y 8.843, Z 72.250} C_DIS
   LIN {X 10.469, Y 3.414, Z 72.250} C_DIS
   LIN {X 10.555, Y 2.020, Z 72.250} C_DIS
   LIN {X 10.660, Y 0.305, Z 72.250} C_DIS
   LIN {X 10.775, Y -3.937, Z 72.250} C_DIS
   LIN {X 10.821, Y -6.208, Z 72.250} C_DIS
   LIN {X 10.743, Y -8.935, Z 72.250} C_DIS
   LIN {X 10.694, Y -10.995, Z 72.250} C_DIS
   LIN {X 10.630, Y -12.041, Z 72.250} C_DIS
   LIN {X 10.445, Y -14.792, Z 72.250} C_DIS
   LIN {X 10.212, Y -17.230, Z 72.250} C_DIS
   LIN {X 10.161, Y -17.740, Z 72.250} C_DIS
   LIN {X 10.028, Y -18.788, Z 72.250} C_DIS
   LIN {X 9.758, Y -20.978, Z 72.250} C_DIS
   LIN {X 9.436, Y -22.016, Z 72.250} C_DIS
   LIN {X 8.870, Y -23.804, Z 72.250} C_DIS
   LIN {X 7.251, Y -26.020, Z 72.250} C_DIS
   LIN {X 7.120, Y -26.201, Z 72.250} C_DIS
   LIN {X 6.969, Y -26.297, Z 72.250} C_DIS
   LIN {X 3.628, Y -28.336, Z 72.250} C_DIS
   LIN {X 1.931, Y -28.621, Z 72.250} C_DIS
   LIN {X 0.517, Y -28.799, Z 72.250} C_DIS
   LIN {X -2.499, Y -28.031, Z 72.250} C_DIS
   LIN {X -3.379, Y -27.794, Z 72.250} C_DIS
   LIN {X -4.350, Y -27.098, Z 72.250} C_DIS
   LIN {X -5.625, Y -26.127, Z 72.250} C_DIS
   LIN {X -6.436, Y -24.857, Z 72.250} C_DIS
   LIN {X -7.563, Y -23.155, Z 72.250} C_DIS
   LIN {X -7.823, Y -21.577, Z 72.250} C_DIS
   LIN {X -8.183, Y -19.497, Z 72.250} C_DIS
   LIN {X -7.536, Y -16.533, Z 72.250} C_DIS
   LIN {X -7.506, Y -16.400, Z 72.250} C_DIS
   LIN {X -7.464, Y -16.295, Z 72.250} C_DIS
   LIN {X -6.269, Y -13.180, Z 72.250} C_DIS
   LIN {X -5.784, Y -11.786, Z 72.250} C_DIS
   LIN {X -5.124, Y -9.517, Z 72.250} C_DIS
   LIN {X -4.423, Y -7.237, Z 72.250} C_DIS
   LIN {X -3.735, Y -4.314, Z 72.250} C_DIS
   LIN {X -3.377, Y -2.693, Z 72.250} C_DIS
   LIN {X -2.393, Y 3.967, Z 72.250} C_DIS
   LIN {X -2.348, Y 4.297, Z 72.250} C_DIS
   LIN {X -2.340, Y 4.521, Z 72.250} C_DIS
   LIN {X -2.240, Y 16.730, Z 72.250} C_DIS
   LIN {X -2.701, Y 21.069, Z 72.250} C_DIS
   LIN {X -3.274, Y 24.842, Z 72.250} C_DIS
   LIN {X -3.670, Y 26.729, Z 72.250} C_DIS
   LIN {X -3.961, Y 28.098, Z 72.250} C_DIS
   LIN {X -4.062, Y 28.461, Z 72.250} C_DIS
   LIN {X -4.126, Y 28.698, Z 72.250} C_DIS
   LIN {X -4.190, Y 28.937, Z 72.250} C_DIS
   LIN {X -5.107, Y 32.368, Z 72.250} C_DIS
   LIN {X -5.722, Y 34.270, Z 72.250} C_DIS
   LIN {X -6.000, Y 35.139, Z 72.250} C_DIS
   LIN {X -6.261, Y 35.861, Z 72.250} C_DIS
   LIN {X -6.809, Y 37.367, Z 72.250} C_DIS
   LIN {X -7.251, Y 38.489, Z 72.250} C_DIS
   LIN {X -7.395, Y 38.856, Z 72.250} C_DIS
   LIN {X -7.480, Y 39.064, Z 72.250} C_DIS
   LIN {X -7.869, Y 40.013, Z 72.250} C_DIS
   LIN {X -8.160, Y 41.176, Z 72.250} C_DIS
   LIN {X -8.187, Y 41.284, Z 72.250} C_DIS
   LIN {X -8.178, Y 41.408, Z 72.250} C_DIS
   LIN {X -8.063, Y 42.609, Z 72.250} C_DIS
   LIN {X -7.363, Y 44.001, Z 72.250} C_DIS
   LIN {X -7.269, Y 44.125, Z 72.250} C_DIS
   LIN {X -6.815, Y 44.572, Z 72.250} C_DIS
   LIN {X -4.993, Y 45.429, Z 72.250}
   LaserEnd_Ext()
   LIN {X 9.602, Y -12.431, Z 72.250}
   LaserStart_Ext()
   LIN {X 9.602, Y 1.221, Z 72.250}
   LaserEnd_Ext()
   LIN {X 8.602, Y 10.377, Z 72.250}
   LaserStart_Ext()
   LIN {X 8.602, Y -21.330, Z 72.250}
   LaserEnd_Ext()
   LIN {X 7.602, Y -23.845, Z 72.250}
   LaserStart_Ext()
   LIN {X 7.602, Y 15.558, Z 72.250}
   LaserEnd_Ext()
   LIN {X 6.602, Y 20.553, Z 72.250}
   LaserStart_Ext()
   LIN {X 6.602, Y -18.430, Z 72.250}
   LaserEnd_Ext()
   LIN {X 6.602, Y -21.040, Z 72.250}
   LaserStart_Ext()
   LIN {X 6.602, Y -25.213, Z 72.250}
   LaserEnd_Ext()
   LIN {X 5.602, Y -25.960, Z 72.250}
   LaserStart_Ext()
   LIN {X 5.602, Y -23.352, Z 72.250}
   LaserEnd_Ext()
   LIN {X 5.602, Y -16.398, Z 72.250}
   LaserStart_Ext()
   LIN {X 5.602, Y 24.351, Z 72.250}
   LaserEnd_Ext()
   LIN {X 4.602, Y 27.572, Z 72.250}
   LaserStart_Ext()
   LIN {X 4.602, Y -15.130, Z 72.250}
   LaserEnd_Ext()
   LIN {X 4.602, Y -24.322, Z 72.250}
   LaserStart_Ext()
   LIN {X 4.602, Y -26.570, Z 72.250}
   LaserEnd_Ext()
   LIN {X 3.602, Y -27.180, Z 72.250}
   LaserStart_Ext()
   LIN {X 3.602, Y -25.037, Z 72.250}
   LaserEnd_Ext()
   LIN {X 3.602, Y -14.572, Z 72.250}
   LaserStart_Ext()
   LIN {X 3.602, Y 30.662, Z 72.250}
   LaserEnd_Ext()
   LIN {X 2.602, Y 33.363, Z 72.250}
   LaserStart_Ext()
   LIN {X 2.602, Y -14.039, Z 72.250}
   LaserEnd_Ext()
   LIN {X 2.602, Y -25.393, Z 72.250}
   LaserStart_Ext()
   LIN {X 2.602, Y -27.494, Z 72.250}
   LaserEnd_Ext()
   LIN {X 1.602, Y -27.654, Z 72.250}
   LaserStart_Ext()
   LIN {X 1.602, Y -25.735, Z 72.250}
   LaserEnd_Ext()
   LIN {X 1.602, Y -13.939, Z 72.250}
   LaserStart_Ext()
   LIN {X 1.602, Y 35.905, Z 72.250}
   LaserEnd_Ext()
   LIN {X 0.602, Y 38.272, Z 72.250}
   LaserStart_Ext()
   LIN {X 0.602, Y -13.862, Z 72.250}
   LaserEnd_Ext()
   LIN {X 0.602, Y -25.694, Z 72.250}
   LaserStart_Ext()
   LIN {X 0.602, Y -27.780, Z 72.250}
   LaserEnd_Ext()
   LIN {X -0.398, Y -27.534, Z 72.250}
   LaserStart_Ext()
   LIN {X -0.398, Y -25.611, Z 72.250}
   LaserEnd_Ext()
   LIN {X -0.398, Y -13.976, Z 72.250}
   LaserStart_Ext()
   LIN {X -0.398, Y 40.504, Z 72.250}
   LaserEnd_Ext()
   LIN {X -1.398, Y 42.610, Z 72.250}
   LaserStart_Ext()
   LIN {X -1.398, Y 18.274, Z 72.250}
   LaserEnd_Ext()
   LIN {X -1.398, Y 3.862, Z 72.250}
   LaserStart_Ext()
   LIN {X -1.398, Y -14.336, Z 72.250}
   LaserEnd_Ext()
   LIN {X -1.398, Y -25.317, Z 72.250}
   LaserStart_Ext()
   LIN {X -1.398, Y -27.279, Z 72.250}
   LaserEnd_Ext()
   LIN {X -2.398, Y -27.022, Z 72.250}
   LaserStart_Ext()
   LIN {X -2.398, Y -24.765, Z 72.250}
   LaserEnd_Ext()
   LIN {X -2.398, Y -14.740, Z 72.250}
   LaserStart_Ext()
   LIN {X -2.398, Y -2.894, Z 72.250}
   LaserEnd_Ext()
   LIN {X -2.398, Y 25.538, Z 72.250}
   LaserStart_Ext()
   LIN {X -2.398, Y 43.855, Z 72.250}
   LaserEnd_Ext()
   LIN {X -3.398, Y 44.401, Z 72.250}
   LaserStart_Ext()
   LIN {X -3.398, Y 29.847, Z 72.250}
   LaserEnd_Ext()
   LIN {X -3.398, Y -7.248, Z 72.250}
   LaserStart_Ext()
   LIN {X -3.398, Y -15.701, Z 72.250}
   LaserEnd_Ext()
   LIN {X -3.398, Y -24.005, Z 72.250}
   LaserStart_Ext()
   LIN {X -3.398, Y -26.549, Z 72.250}
   LaserEnd_Ext()
   LIN {X -4.398, Y -25.804, Z 72.250}
   LaserStart_Ext()
   LIN {X -4.398, Y -22.690, Z 72.250}
   LaserEnd_Ext()
   LIN {X -4.398, Y -17.118, Z 72.250}
   LaserStart_Ext()
   LIN {X -4.398, Y -10.601, Z 72.250}
   LaserEnd_Ext()
   LIN {X -4.398, Y 33.426, Z 72.250}
   LaserStart_Ext()
   LIN {X -4.398, Y 44.490, Z 72.250}
   LaserEnd_Ext()
   LIN {X -5.398, Y 44.133, Z 72.250}
   LaserStart_Ext()
   LIN {X -5.398, Y 36.413, Z 72.250}
   LaserEnd_Ext()
   LIN {X -5.398, Y -13.701, Z 72.250}
   LaserStart_Ext()
   LIN {X -5.398, Y -24.625, Z 72.250}
   LaserEnd_Ext()
   LIN {X -6.398, Y -23.103, Z 72.250}
   LaserStart_Ext()
   LIN {X -6.398, Y -16.307, Z 72.250}
   LaserEnd_Ext()
   LIN {X -6.398, Y 39.052, Z 72.250}
   LaserStart_Ext()
   LIN {X -6.398, Y 43.579, Z 72.250}
   LaserEnd_Ext()
   LIN {X 3.567, Y -23.959, Z 73.100}
   LaserStart_Ext()
   LIN {X 1.624, Y -24.654, Z 73.100} C_DIS
   LIN {X 1.492, Y -24.701, Z 73.100} C_DIS
   LIN {X -0.557, Y -24.537, Z 73.100} C_DIS
   LIN {X -1.927, Y -23.788, Z 73.100} C_DIS
   LIN {X -2.369, Y -23.544, Z 73.100} C_DIS
   LIN {X -2.764, Y -23.025, Z 73.100} C_DIS
   LIN {X -3.633, Y -21.888, Z 73.100} C_DIS
   LIN {X -3.962, Y -20.461, Z 73.100} C_DIS
   LIN {X -4.099, Y -19.855, Z 73.100} C_DIS
   LIN {X -3.976, Y -19.448, Z 73.100} C_DIS
   LIN {X -3.272, Y -17.007, Z 73.100} C_DIS
   LIN {X -2.851, Y -16.597, Z 73.100} C_DIS
   LIN {X -1.784, Y -15.529, Z 73.100} C_DIS
   LIN {X 0.034, Y -14.845, Z 73.100} C_DIS
   LIN {X 0.202, Y -14.785, Z 73.100} C_DIS
   LIN {X 0.341, Y -14.796, Z 73.100} C_DIS
   LIN {X 2.358, Y -14.930, Z 73.100} C_DIS
   LIN {X 4.013, Y -15.847, Z 73.100} C_DIS
   LIN {X 4.217, Y -15.959, Z 73.100} C_DIS
   LIN {X 4.377, Y -16.194, Z 73.100} C_DIS
   LIN {X 5.639, Y -18.067, Z 73.100} C_DIS
   LIN {X 5.875, Y -20.220, Z 73.100} C_DIS
   LIN {X 5.843, Y -20.365, Z 73.100} C_DIS
   LIN {X 5.046, Y -22.517, Z 73.100} C_DIS
   LIN {X 4.429, Y -23.122, Z 73.100} C_DIS
   LIN {X 3.567, Y -23.959, Z 73.100}
   LaserEnd_Ext()
   LIN {X 4.209, Y 31.831, Z 73.100}
   LaserStart_Ext()
   LIN {X 3.103, Y 34.818, Z 73.100} C_DIS
   LIN {X 3.005, Y 35.052, Z 73.100} C_DIS
   LIN {X 1.888, Y 37.770, Z 73.100} C_DIS
   LIN {X 1.125, Y 39.481, Z 73.100} C_DIS
   LIN {X 0.765, Y 40.298, Z 73.100} C_DIS
   LIN {X 0.052, Y 41.819, Z 73.100} C_DIS
   LIN {X -0.049, Y 42.033, Z 73.100} C_DIS
   LIN {X -0.154, Y 42.248, Z 73.100} C_DIS
   LIN {X -0.698, Y 43.367, Z 73.100} C_DIS
   LIN {X -1.333, Y 44.213, Z 73.100} C_DIS
   LIN {X -1.582, Y 44.544, Z 73.100} C_DIS
   LIN {X -2.238, Y 44.923, Z 73.100} C_DIS
   LIN {X -3.088, Y 45.416, Z 73.100} C_DIS
   LIN {X -3.637, Y 45.464, Z 73.100} C_DIS
   LIN {X -4.826, Y 45.566, Z 73.100} C_DIS
   LIN {X -6.188, Y 44.816, Z 73.100} C_DIS
   LIN {X -7.137, Y 44.370, Z 73.100} C_DIS
   LIN {X -7.352, Y 44.158, Z 73.100} C_DIS
   LIN {X -7.967, Y 42.915, Z 73.100} C_DIS
   LIN {X -8.158, Y 42.544, Z 73.100} C_DIS
   LIN {X -8.181, Y 42.241, Z 73.100} C_DIS
   LIN {X -8.249, Y 41.296, Z 73.100} C_DIS
   LIN {X -7.959, Y 40.158, Z 73.100} C_DIS
   LIN {X -7.930, Y 40.046, Z 73.100} C_DIS
   LIN {X -7.453, Y 38.890, Z 73.100} C_DIS
   LIN {X -6.987, Y 37.717, Z 73.100} C_DIS
   LIN {X -6.863, Y 37.403, Z 73.100} C_DIS
   LIN {X -6.676, Y 36.888, Z 73.100} C_DIS
   LIN {X -6.050, Y 35.177, Z 73.100} C_DIS
   LIN {X -5.407, Y 33.205, Z 73.100} C_DIS
   LIN {X -5.150, Y 32.408, Z 73.100} C_DIS
   LIN {X -4.986, Y 31.793, Z 73.100} C_DIS
   LIN {X -4.519, Y 30.050, Z 73.100} C_DIS
   LIN {X -4.359, Y 29.452, Z 73.100} C_DIS
   LIN {X -4.232, Y 28.975, Z 73.100} C_DIS
   LIN {X -4.200, Y 28.856, Z 73.100} C_DIS
   LIN {X -3.946, Y 27.948, Z 73.100} C_DIS
   LIN {X -3.332, Y 25.065, Z 73.100} C_DIS
   LIN {X -3.262, Y 24.608, Z 73.100} C_DIS
   LIN {X -2.619, Y 20.377, Z 73.100} C_DIS
   LIN {X -2.255, Y 16.946, Z 73.100} C_DIS
   LIN {X -2.343, Y 6.154, Z 73.100} C_DIS
   LIN {X -2.322, Y 4.543, Z 73.100} C_DIS
   LIN {X -2.361, Y 3.997, Z 73.100} C_DIS
   LIN {X -3.085, Y -0.801, Z 73.100} C_DIS
   LIN {X -3.420, Y -3.073, Z 73.100} C_DIS
   LIN {X -3.502, Y -3.443, Z 73.100} C_DIS
   LIN {X -4.481, Y -7.601, Z 73.100} C_DIS
   LIN {X -5.479, Y -10.845, Z 73.100} C_DIS
   LIN {X -5.857, Y -12.146, Z 73.100} C_DIS
   LIN {X -6.135, Y -12.945, Z 73.100} C_DIS
   LIN {X -6.874, Y -14.870, Z 73.100} C_DIS
   LIN {X -7.434, Y -16.365, Z 73.100} C_DIS
   LIN {X -7.622, Y -17.257, Z 73.100} C_DIS
   LIN {X -8.105, Y -19.464, Z 73.100} C_DIS
   LIN {X -7.554, Y -22.648, Z 73.100} C_DIS
   LIN {X -7.476, Y -23.121, Z 73.100} C_DIS
   LIN {X -7.138, Y -23.631, Z 73.100} C_DIS
   LIN {X -5.649, Y -25.963, Z 73.100} C_DIS
   LIN {X -3.389, Y -27.683, Z 73.100} C_DIS
   LIN {X -2.839, Y -27.843, Z 73.100} C_DIS
   LIN {X 0.719, Y -28.749, Z 73.100} C_DIS
   LIN {X 1.048, Y -28.708, Z 73.100} C_DIS
   LIN {X 3.824, Y -28.242, Z 73.100} C_DIS
   LIN {X 5.811, Y -27.030, Z 73.100} C_DIS
   LIN {X 7.214, Y -26.132, Z 73.100} C_DIS
   LIN {X 8.437, Y -24.445, Z 73.100} C_DIS
   LIN {X 8.959, Y -23.731, Z 73.100} C_DIS
   LIN {X 9.142, Y -23.154, Z 73.100} C_DIS
   LIN {X 9.840, Y -20.903, Z 73.100} C_DIS
   LIN {X 10.152, Y -18.375, Z 73.100} C_DIS
   LIN {X 10.235, Y -17.663, Z 73.100} C_DIS
   LIN {X 10.327, Y -16.659, Z 73.100} C_DIS
   LIN {X 10.513, Y -14.715, Z 73.100} C_DIS
   LIN {X 10.612, Y -13.248, Z 73.100} C_DIS
   LIN {X 10.752, Y -10.917, Z 73.100} C_DIS
   LIN {X 10.862, Y -6.331, Z 73.100} C_DIS
   LIN {X 10.868, Y -6.131, Z 73.100} C_DIS
   LIN {X 10.865, Y -5.964, Z 73.100} C_DIS
   LIN {X 10.692, Y 0.383, Z 73.100} C_DIS
   LIN {X 10.618, Y 1.587, Z 73.100} C_DIS
   LIN {X 10.523, Y 3.130, Z 73.100} C_DIS
   LIN {X 9.845, Y 9.138, Z 73.100} C_DIS
   LIN {X 9.808, Y 9.376, Z 73.100} C_DIS
   LIN {X 7.674, Y 20.429, Z 73.100} C_DIS
   LIN {X 6.549, Y 24.703, Z 73.100} C_DIS
   LIN {X 5.044, Y 29.409, Z 73.100} C_DIS
   LIN {X 4.628, Y 30.739, Z 73.100} C_DIS
   LIN {X 4.209, Y 31.831, Z 73.100}
   LaserEnd_Ext()
   LIN {X -4.350, Y 44.522, Z 73.100}
   LaserStart_Ext()
   LIN {X -4.650, Y 44.522, Z 73.100}
   LaserEnd_Ext()
   LIN {X -6.551, Y 43.522, Z 73.100}
   LaserStart_Ext()
   LIN {X -2.064, Y 43.522, Z 73.100}
   LaserEnd_Ext()
   LIN {X -1.399, Y 42.522, Z 73.100}
   LaserStart_Ext()
   LIN {X -7.046, Y 42.522, Z 73.100}
   LaserEnd_Ext()
   LIN {X -7.230, Y 41.522, Z 73.100}
   LaserStart_Ext()
   LIN {X -0.913, Y 41.522, Z 73.100}
   LaserEnd_Ext()
   LIN {X -0.444, Y 40.522, Z 73.100}
   LaserStart_Ext()
   LIN {X -7.020, Y 40.522, Z 73.100}
   LaserEnd_Ext()
   LIN {X -6.632, Y 39.522, Z 73.100}
   LaserStart_Ext()
   LIN {X 0.014, Y 39.522, Z 73.100}
   LaserEnd_Ext()
   LIN {X 0.458, Y 38.522, Z 73.100}
   LaserStart_Ext()
   LIN {X -6.231, Y 38.522, Z 73.100}
   LaserEnd_Ext()
   LIN {X -5.842, Y 37.522, Z 73.100}
   LaserStart_Ext()
   LIN {X 0.903, Y 37.522, Z 73.100}
   LaserEnd_Ext()
   LIN {X 1.320, Y 36.522, Z 73.100}
   LaserStart_Ext()
   LIN {X -5.477, Y 36.522, Z 73.100}
   LaserEnd_Ext()
   LIN {X -5.111, Y 35.522, Z 73.100}
   LaserStart_Ext()
   LIN {X 1.731, Y 35.522, Z 73.100}
   LaserEnd_Ext()
   LIN {X 2.143, Y 34.522, Z 73.100}
   LaserStart_Ext()
   LIN {X -4.785, Y 34.522, Z 73.100}
   LaserEnd_Ext()
   LIN {X -4.459, Y 33.522, Z 73.100}
   LaserStart_Ext()
   LIN {X 2.516, Y 33.522, Z 73.100}
   LaserEnd_Ext()
   LIN {X 2.887, Y 32.522, Z 73.100}
   LaserStart_Ext()
   LIN {X -4.145, Y 32.522, Z 73.100}
   LaserEnd_Ext()
   LIN {X -3.878, Y 31.522, Z 73.100}
   LaserStart_Ext()
   LIN {X 3.258, Y 31.522, Z 73.100}
   LaserEnd_Ext()
   LIN {X 3.640, Y 30.522, Z 73.100}
   LaserStart_Ext()
   LIN {X -3.610, Y 30.522, Z 73.100}
   LaserEnd_Ext()
   LIN {X -3.343, Y 29.522, Z 73.100}
   LaserStart_Ext()
   LIN {X 3.961, Y 29.522, Z 73.100}
   LaserEnd_Ext()
   LIN {X 4.278, Y 28.522, Z 73.100}
   LaserStart_Ext()
   LIN {X -3.068, Y 28.522, Z 73.100}
   LaserEnd_Ext()
   LIN {X -2.833, Y 27.522, Z 73.100}
   LaserStart_Ext()
   LIN {X 4.598, Y 27.522, Z 73.100}
   LaserEnd_Ext()
   LIN {X 4.918, Y 26.522, Z 73.100}
   LaserStart_Ext()
   LIN {X -2.620, Y 26.522, Z 73.100}
   LaserEnd_Ext()
   LIN {X -2.407, Y 25.522, Z 73.100}
   LaserStart_Ext()
   LIN {X 5.237, Y 25.522, Z 73.100}
   LaserEnd_Ext()
   LIN {X 5.557, Y 24.522, Z 73.100}
   LaserStart_Ext()
   LIN {X -2.237, Y 24.522, Z 73.100}
   LaserEnd_Ext()
   LIN {X -2.085, Y 23.522, Z 73.100}
   LaserStart_Ext()
   LIN {X 5.826, Y 23.522, Z 73.100}
   LaserEnd_Ext()
   LIN {X 6.089, Y 22.522, Z 73.100}
   LaserStart_Ext()
   LIN {X -1.933, Y 22.522, Z 73.100}
   LaserEnd_Ext()
   LIN {X -1.781, Y 21.522, Z 73.100}
   LaserStart_Ext()
   LIN {X 6.353, Y 21.522, Z 73.100}
   LaserEnd_Ext()
   LIN {X 6.616, Y 20.522, Z 73.100}
   LaserStart_Ext()
   LIN {X -1.630, Y 20.522, Z 73.100}
   LaserEnd_Ext()
   LIN {X -1.522, Y 19.522, Z 73.100}
   LaserStart_Ext()
   LIN {X 6.831, Y 19.522, Z 73.100}
   LaserEnd_Ext()
   LIN {X 7.024, Y 18.522, Z 73.100}
   LaserStart_Ext()
   LIN {X -1.416, Y 18.522, Z 73.100}
   LaserEnd_Ext()
   LIN {X -1.310, Y 17.522, Z 73.100}
   LaserStart_Ext()
   LIN {X 7.217, Y 17.522, Z 73.100}
   LaserEnd_Ext()
   LIN {X 7.410, Y 16.522, Z 73.100}
   LaserStart_Ext()
   LIN {X -1.258, Y 16.522, Z 73.100}
   LaserEnd_Ext()
   LIN {X -1.266, Y 15.522, Z 73.100}
   LaserStart_Ext()
   LIN {X 7.603, Y 15.522, Z 73.100}
   LaserEnd_Ext()
   LIN {X 7.796, Y 14.522, Z 73.100}
   LaserStart_Ext()
   LIN {X -1.274, Y 14.522, Z 73.100}
   LaserEnd_Ext()
   LIN {X -1.283, Y 13.522, Z 73.100}
   LaserStart_Ext()
   LIN {X 7.989, Y 13.522, Z 73.100}
   LaserEnd_Ext()
   LIN {X 8.182, Y 12.522, Z 73.100}
   LaserStart_Ext()
   LIN {X -1.291, Y 12.522, Z 73.100}
   LaserEnd_Ext()
   LIN {X -1.299, Y 11.522, Z 73.100}
   LaserStart_Ext()
   LIN {X 8.375, Y 11.522, Z 73.100}
   LaserEnd_Ext()
   LIN {X 8.568, Y 10.522, Z 73.100}
   LaserStart_Ext()
   LIN {X -1.307, Y 10.522, Z 73.100}
   LaserEnd_Ext()
   LIN {X -1.315, Y 9.522, Z 73.100}
   LaserStart_Ext()
   LIN {X 8.761, Y 9.522, Z 73.100}
   LaserEnd_Ext()
   LIN {X 8.908, Y 8.522, Z 73.100}
   LaserStart_Ext()
   LIN {X -1.324, Y 8.522, Z 73.100}
   LaserEnd_Ext()
   LIN {X -1.332, Y 7.522, Z 73.100}
   LaserStart_Ext()
   LIN {X 9.021, Y 7.522, Z 73.100}
   LaserEnd_Ext()
   LIN {X 9.134, Y 6.522, Z 73.100}
   LaserStart_Ext()
   LIN {X -1.340, Y 6.522, Z 73.100}
   LaserEnd_Ext()
   LIN {X -1.335, Y 5.522, Z 73.100}
   LaserStart_Ext()
   LIN {X 9.247, Y 5.522, Z 73.100}
   LaserEnd_Ext()
   LIN {X 9.360, Y 4.522, Z 73.100}
   LaserStart_Ext()
   LIN {X -1.324, Y 4.522, Z 73.100}
   LaserEnd_Ext()
   LIN {X -1.422, Y 3.522, Z 73.100}
   LaserStart_Ext()
   LIN {X 9.473, Y 3.522, Z 73.100}
   LaserEnd_Ext()
   LIN {X 9.559, Y 2.522, Z 73.100}
   LaserStart_Ext()
   LIN {X -1.572, Y 2.522, Z 73.100}
   LaserEnd_Ext()
   LIN {X -1.723, Y 1.522, Z 73.100}
   LaserStart_Ext()
   LIN {X 9.620, Y 1.522, Z 73.100}
   LaserEnd_Ext()
